// TIA Portal V16 program export: 0 tag tables, 0 data types, 2 data blocks, 11 code blocks (in call order from the OBs), 4 instance data blocks

DATA_BLOCK "DB_HMI"   // DB3
{ S7_Optimized_Access := 'TRUE' }
VERSION : 0.1
// stored: AutoNumber true, CodeModifiedDate 2020-02-26T07:38:35.2363514Z, CompileDate 2021-07-03T08:38:43.1466981Z, CreationDate 2020-02-26T07:38:17.5478271Z, DBAccessibleFromOPCUA true, DownloadWithoutReinit false, InterfaceModifiedDate 2020-02-26T07:38:35.2363514Z, IsConsistent true, IsKnowHowProtected false, IsOnlyStoredInLoadMemory false, IsPLCDB false, IsRetainMemResEnabled false, IsWriteProtectedInAS false, MemoryReserve 100, ModifiedDate 2020-02-26T07:38:35.2363514Z, ParameterModified 2020-02-26T07:38:35.2363514Z, StructureModified 2020-02-26T07:38:35.2363514Z
   VAR
      VlvLiq1 : "udtHMI_ValveControl";
      VlvLiq2 { S7_SetPoint := 'True'} : "udtHMI_ValveControl";
      VlvDrn { S7_SetPoint := 'True'} : "udtHMI_ValveControl";
   END_VAR
BEGIN
END_DATA_BLOCK

DATA_BLOCK "DB_ProgramLogic"   // DB4
{ S7_Optimized_Access := 'TRUE' }
VERSION : 0.1
// stored: AutoNumber true, CodeModifiedDate 2020-02-26T07:40:10.2847553Z, CompileDate 2021-07-03T08:38:37.7718266Z, CreationDate 2020-02-26T07:39:28.2364137Z, DBAccessibleFromOPCUA true, DownloadWithoutReinit false, InterfaceModifiedDate 2020-02-26T07:40:10.2847553Z, IsConsistent true, IsKnowHowProtected false, IsOnlyStoredInLoadMemory false, IsPLCDB false, IsRetainMemResEnabled false, IsWriteProtectedInAS false, MemoryReserve 100, ModifiedDate 2020-02-26T07:40:10.2847553Z, ParameterModified 2020-02-26T07:40:10.2847553Z, StructureModified 2020-02-26T07:40:10.2847553Z
   VAR
      VlvLiq1_Open : Bool;
      VlvLiq2_Open : Bool;
      VlvDrn_Open : Bool;
   END_VAR
BEGIN
END_DATA_BLOCK

ORGANIZATION_BLOCK "Main"   // OB1, FBD, ProgramCycle
TITLE = "Main Program Sweep (Cycle)"
{ S7_Optimized_Access := 'TRUE' }
VERSION : 0.1
// stored: AutoNumber true, CodeModifiedDate 2021-08-10T08:54:10.1985647Z, CompileDate 2021-08-10T08:57:18.4266346Z, ConstantName OB_Main, CreationDate 2020-02-26T07:01:34.5488912Z, EventClass Program cycle, HandleErrorsWithinBlock false, InterfaceModifiedDate 2008-07-21T16:55:08.419547Z, IsConsistent true, IsIECCheckEnabled false, IsKnowHowProtected false, IsWriteProtected false, ModifiedDate 2021-08-10T08:54:10.1985647Z, ParameterModified 2008-07-21T16:55:08.419547Z, PLCSimAdvancedSupport true, PriorityNumber 1, ProcessImagePartNumber 65535, SetENOAutomatically false, StructureModified 2008-07-21T16:55:08.419547Z
   VAR_INPUT
      Initial_Call : Bool;   // Initial call of this OB
      Remanence : Bool;   // =True, if remanent data are available
   END_VAR
BEGIN

REGION Network 1
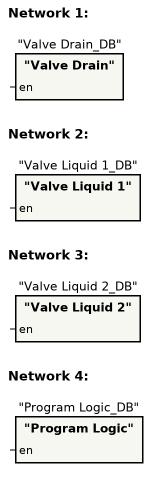
   "Valve Drain_DB"();   // "Valve Drain"
END_REGION

REGION Network 2
   "Valve Liquid 1_DB"();   // "Valve Liquid 1"
END_REGION

REGION Network 3
   "Valve Liquid 2_DB"();   // "Valve Liquid 2"
END_REGION

REGION Network 4
   "Program Logic_DB"();   // "Program Logic"
END_REGION
END_ORGANIZATION_BLOCK

FUNCTION_BLOCK "Valve Drain"   // FB4, FBD
{ S7_Optimized_Access := 'TRUE' }
VERSION : 0.1
// stored: AutoNumber true, CodeModifiedDate 2020-02-26T13:08:47.8951368Z, CompileDate 2021-07-03T08:38:43.4907825Z, CreationDate 2020-02-26T07:16:51.9541274Z, DownloadWithoutReinit false, HandleErrorsWithinBlock false, InterfaceModifiedDate 2020-02-26T12:48:59.514304Z, IsConsistent true, IsIECCheckEnabled false, IsKnowHowProtected false, ISMultiInstanceCapable true, IsRetainMemResEnabled false, IsWriteProtected false, LibraryConformanceStatus Warning: The object contains access to global data blocks. Warning: The block contains direct access to inputs, outputs, bit memories, indirect access to the registry or indirect access to external memory areas that are unknown at the time of compilation., MemoryReserve 100, ModifiedDate 2020-05-11T19:30:06.5567173Z, ParameterModified 2020-02-26T07:16:51.9541274Z, PLCSimAdvancedSupport true, SetENOAutomatically false, StructureModified 2020-02-26T12:48:59.514304Z, UDAEnableTagReadback false
   VAR
      VlvDrn : "fbValve_Solenoid";
   END_VAR
BEGIN

REGION Network 1
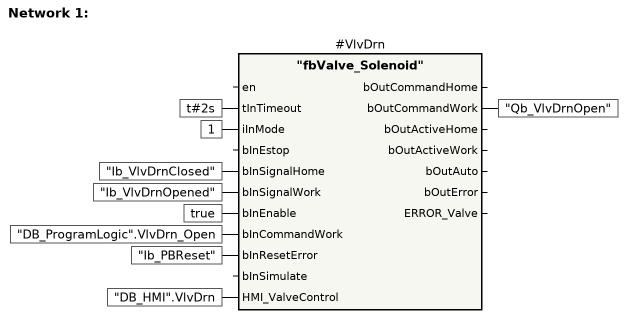
   #VlvDrn(tInTimeout := t#2s,   // "fbValve_Solenoid"
           iInMode := 1,
           bInSignalHome := "Ib_VlvDrnClosed",
           bInSignalWork := "Ib_VlvDrnOpened",
           bInEnable := true,
           bInCommandWork := "DB_ProgramLogic".VlvDrn_Open,
           bInResetError := "Ib_PBReset",
           HMI_ValveControl := "DB_HMI".VlvDrn,
           bOutCommandWork => "Qb_VlvDrnOpen");
END_REGION
END_FUNCTION_BLOCK

FUNCTION_BLOCK "fbValve_Solenoid"   // FB110, FBD
TITLE = Controls a double- or single-acting valve
{ S7_Optimized_Access := 'TRUE' }
VERSION : 0.1
// stored: AutoNumber false, CodeModifiedDate 2021-08-10T11:52:58.0273326Z, CompileDate 2021-08-10T11:53:23.0999729Z, CreationDate 2020-02-26T07:34:28.9567791Z, DownloadWithoutReinit false, HandleErrorsWithinBlock false, InterfaceModifiedDate 2019-07-17T06:42:37.7805928Z, IsConsistent true, IsIECCheckEnabled false, IsKnowHowProtected false, ISMultiInstanceCapable true, IsRetainMemResEnabled false, IsWriteProtected false, LibraryConformanceStatus Warning: The object contains access to global PLC constants., LibraryType fbValve_Solenoid V 3.0.6 in test, LibraryTypeVersionGuid 0a9fd967-cd2b-46e1-afc3-82055bb762c7, MemoryReserve 100, ModifiedDate 2021-08-10T11:52:58.0273326Z, ParameterModified 2019-07-17T06:42:37.7805928Z, PLCSimAdvancedSupport true, SetENOAutomatically false, StructureModified 2019-07-17T06:42:37.7805928Z, UDAEnableTagReadback false
   VAR_INPUT
      tInTimeout { ExternalAccessible := 'False'; ExternalVisible := 'False'; ExternalWritable := 'False'} : Time;   // Timeout time for an actuator's feedback to activate before giving a fault
      iInMode { ExternalAccessible := 'False'; ExternalVisible := 'False'; ExternalWritable := 'False'} : Int;   // Mode Selection
      bInEstop { ExternalAccessible := 'False'; ExternalVisible := 'False'; ExternalWritable := 'False'} : Bool;   // Estop
      bInSignalHome { ExternalAccessible := 'False'; ExternalVisible := 'False'; ExternalWritable := 'False'} : Bool;   // Home position feedback
      bInSignalWork { ExternalAccessible := 'False'; ExternalVisible := 'False'; ExternalWritable := 'False'} : Bool;   // Work position feedback
      bInEnable { ExternalAccessible := 'False'; ExternalVisible := 'False'; ExternalWritable := 'False'} : Bool;   // Home and Work Enabled
      bInCommandWork { ExternalAccessible := 'False'; ExternalVisible := 'False'; ExternalWritable := 'False'} : Bool;   // Move to work position in automatic mode
      bInResetError { ExternalAccessible := 'False'; ExternalVisible := 'False'; ExternalWritable := 'False'} : Bool;   // Reset Error
      bInSimulate { ExternalAccessible := 'False'; ExternalVisible := 'False'; ExternalWritable := 'False'} : Bool;   // Activate device simulation
   END_VAR
   VAR_OUTPUT
      bOutCommandHome { ExternalAccessible := 'False'; ExternalVisible := 'False'; ExternalWritable := 'False'} : Bool;   // Home position command
      bOutCommandWork { ExternalAccessible := 'False'; ExternalVisible := 'False'; ExternalWritable := 'False'} : Bool;   // Work position command
      bOutActiveHome { ExternalAccessible := 'False'; ExternalVisible := 'False'; ExternalWritable := 'False'} : Bool;   // Valve is in home position
      bOutActiveWork { ExternalAccessible := 'False'; ExternalVisible := 'False'; ExternalWritable := 'False'} : Bool;   // Valve is in work position
      bOutAuto { ExternalAccessible := 'False'; ExternalVisible := 'False'; ExternalWritable := 'False'} : Bool;   // Block in auto mode
      bOutError { ExternalAccessible := 'False'; ExternalVisible := 'False'; ExternalWritable := 'False'} : Bool;   // Error exists
      ERROR_Valve { ExternalAccessible := 'False'; ExternalVisible := 'False'; ExternalWritable := 'False'} : "udtError_Valve";   // Valve error structure
   END_VAR
   VAR_IN_OUT
      HMI_ValveControl : "udtHMI_ValveControl";   // HMI valve control
   END_VAR
   VAR
      ErrorScroller { ExternalAccessible := 'False'; ExternalVisible := 'False'; ExternalWritable := 'False'; S7_SetPoint := 'True'} : "fbErrorScroller";   // Sub-block to handle error scroller
      TON_TimeOut { ExternalAccessible := 'False'; ExternalVisible := 'False'; ExternalWritable := 'False'; S7_SetPoint := 'True'} : TON_TIME;   // Timer for Error Timeout
      iLastMode { ExternalAccessible := 'False'; ExternalVisible := 'False'; ExternalWritable := 'False'} : Int;   // Last mode code
      bNewMode { ExternalAccessible := 'False'; ExternalVisible := 'False'; ExternalWritable := 'False'} : Bool;   // New mode selected
      bEnableHome { ExternalAccessible := 'False'; ExternalVisible := 'False'; ExternalWritable := 'False'} : Bool;   // Home position enabled
      bEnableWork { ExternalAccessible := 'False'; ExternalVisible := 'False'; ExternalWritable := 'False'} : Bool;   // Work position enabled
      bAutoMode { ExternalAccessible := 'False'; ExternalVisible := 'False'; ExternalWritable := 'False'} : Bool;   // Auto Mode is active
      bManualMode { ExternalAccessible := 'False'; ExternalVisible := 'False'; ExternalWritable := 'False'} : Bool;   // Manual Mode is active
      bReset { ExternalAccessible := 'False'; ExternalVisible := 'False'; ExternalWritable := 'False'} : Bool;
      bTON_TimeOut { ExternalAccessible := 'False'; ExternalVisible := 'False'; ExternalWritable := 'False'} : Bool;
      bPB_Home { ExternalAccessible := 'False'; ExternalVisible := 'False'; ExternalWritable := 'False'} : Bool;
      bPB_Work { ExternalAccessible := 'False'; ExternalVisible := 'False'; ExternalWritable := 'False'} : Bool;
      bPB_ResetError { ExternalAccessible := 'False'; ExternalVisible := 'False'; ExternalWritable := 'False'} : Bool;
   END_VAR
   VAR_TEMP
      tTimeoutElapsed : Time;   // Elapsed time for TON_Timeout
      bTemp : Bool;
   END_VAR
   VAR_TEMP   // added for the SCL form of the ladder/FBD networks
      _w1 : Bool;
      _w2 : Bool;
   END_VAR
BEGIN

REGION Network 1: --------------------------------------------------------- Inputs ------------------------------------------------------------------
END_REGION

REGION Network 2: Read HMI input buttons
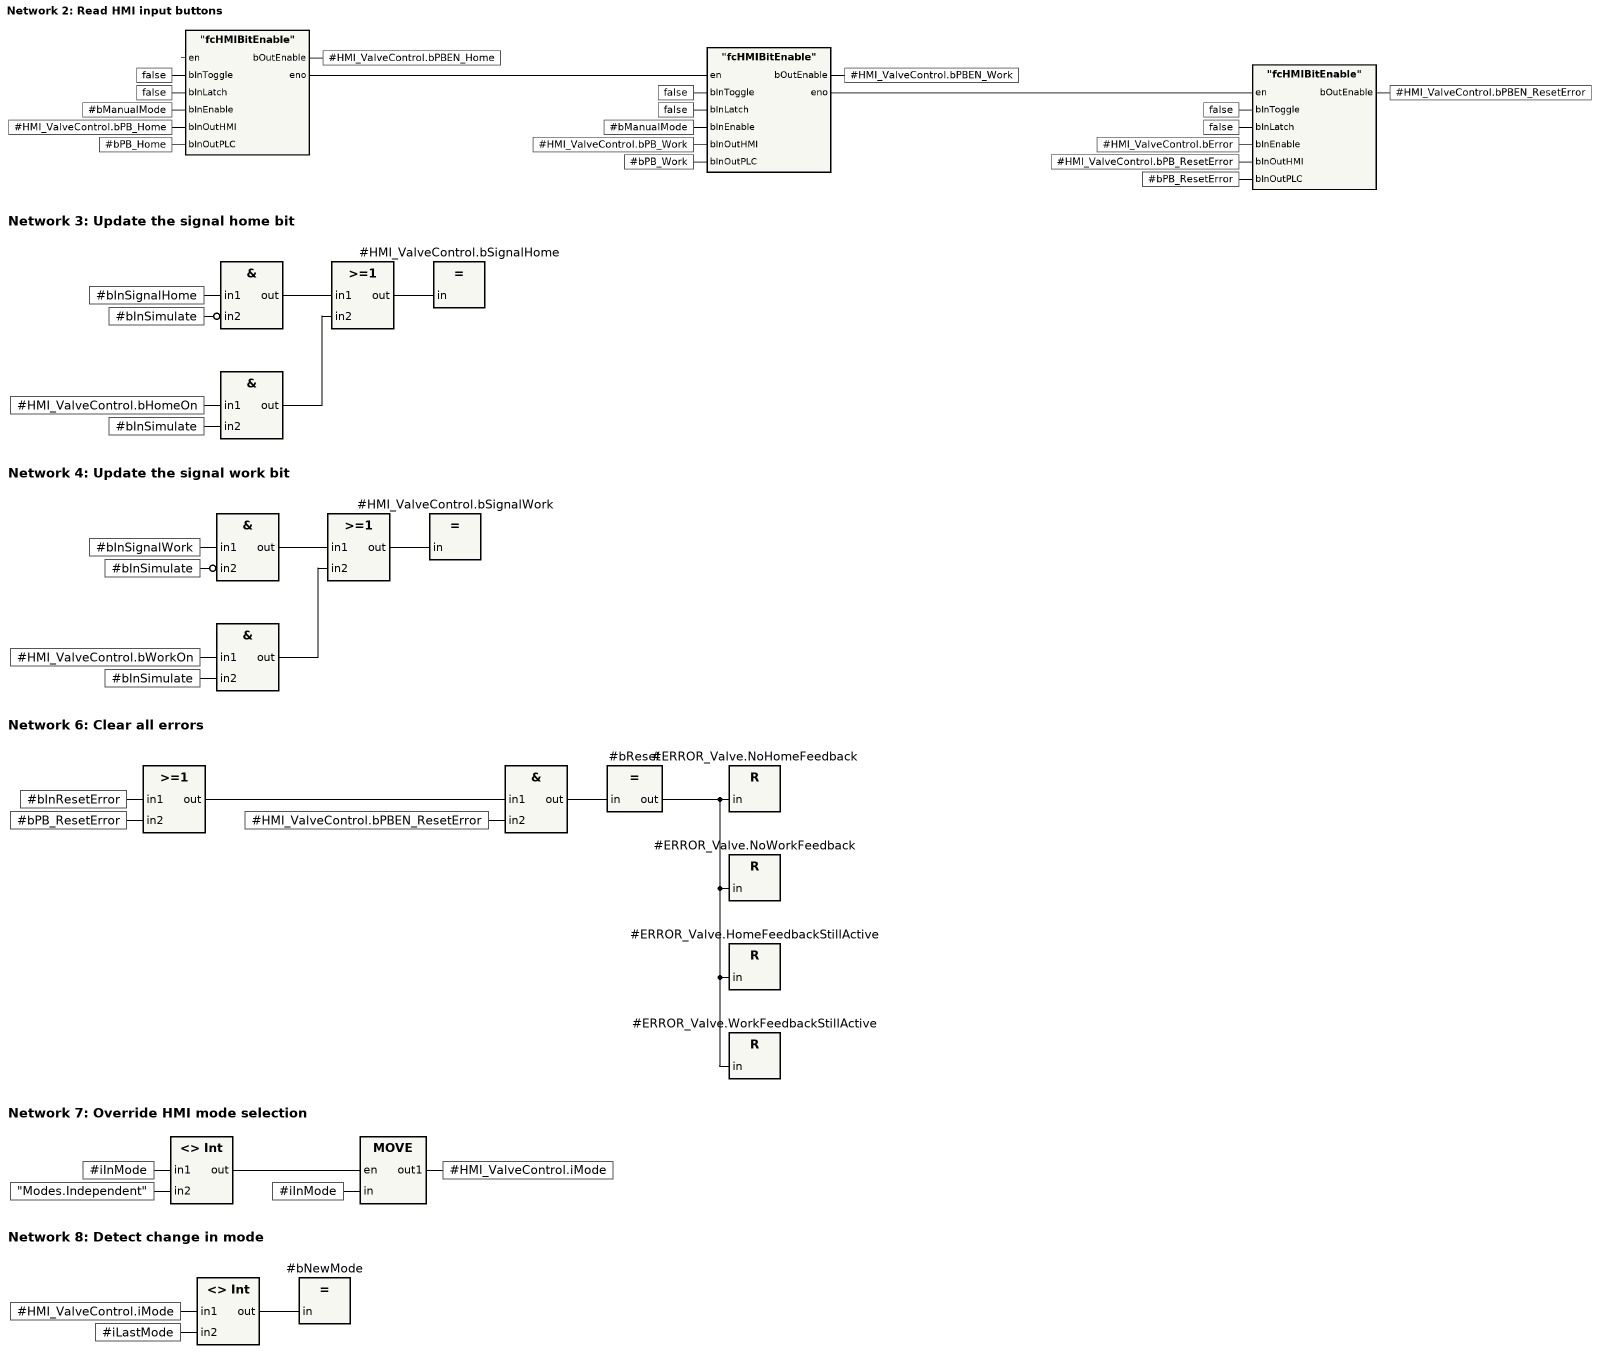
   "fcHMIBitEnable"(bInToggle := false,
                    bInLatch := false,
                    bInEnable := #bManualMode,
                    bInOutHMI := #HMI_ValveControl.bPB_Home,
                    bInOutPLC := #bPB_Home,
                    bOutEnable => #HMI_ValveControl.bPBEN_Home,
                    ENO => #_w1);
   "fcHMIBitEnable"(EN := #_w1,
                    bInToggle := false,
                    bInLatch := false,
                    bInEnable := #bManualMode,
                    bInOutHMI := #HMI_ValveControl.bPB_Work,
                    bInOutPLC := #bPB_Work,
                    bOutEnable => #HMI_ValveControl.bPBEN_Work,
                    ENO => #_w2);
   IF #_w2 THEN
       "fcHMIBitEnable"(bInToggle := false,
                        bInLatch := false,
                        bInEnable := #HMI_ValveControl.bError,
                        bInOutHMI := #HMI_ValveControl.bPB_ResetError,
                        bInOutPLC := #bPB_ResetError,
                        bOutEnable => #HMI_ValveControl.bPBEN_ResetError);
   END_IF;
END_REGION

REGION Network 3: Update the signal home bit
   #HMI_ValveControl.bSignalHome := (#bInSignalHome AND NOT #bInSimulate) OR (#HMI_ValveControl.bHomeOn AND #bInSimulate);
END_REGION

REGION Network 4: Update the signal work bit
   #HMI_ValveControl.bSignalWork := (#bInSignalWork AND NOT #bInSimulate) OR (#HMI_ValveControl.bWorkOn AND #bInSimulate);
END_REGION

REGION Network 5: --------------------------------------------------- Control Logic ------------------------------------------------------------
END_REGION

REGION Network 6: Clear all errors
   #bReset := (#bInResetError OR #bPB_ResetError) AND #HMI_ValveControl.bPBEN_ResetError;
   IF #bReset THEN
       #ERROR_Valve.NoHomeFeedback := FALSE;
       #ERROR_Valve.NoWorkFeedback := FALSE;
       #ERROR_Valve.HomeFeedbackStillActive := FALSE;
       #ERROR_Valve.WorkFeedbackStillActive := FALSE;
   END_IF;
END_REGION

REGION Network 7: Override HMI mode selection
   IF #iInMode <> "Modes.Independent" THEN #HMI_ValveControl.iMode := #iInMode; END_IF;
END_REGION

REGION Network 8: Detect change in mode
   #bNewMode := #HMI_ValveControl.iMode <> #iLastMode;
END_REGION

REGION Network 9: Keep track of last mode
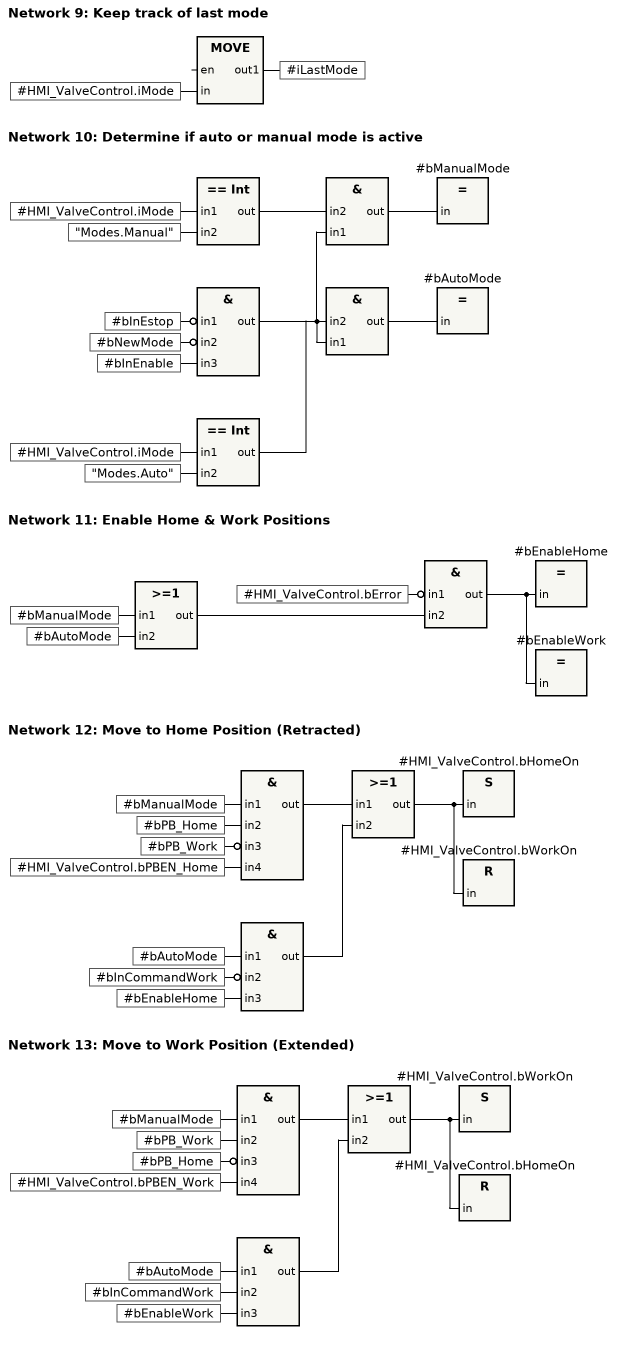
   #iLastMode := #HMI_ValveControl.iMode;
END_REGION

REGION Network 10: Determine if auto or manual mode is active
   #_w1 := NOT #bInEstop AND NOT #bNewMode AND #bInEnable;
   #bManualMode := (#HMI_ValveControl.iMode = "Modes.Manual") AND #_w1;
   #bAutoMode := (#HMI_ValveControl.iMode = "Modes.Auto") AND #_w1;
END_REGION

REGION Network 11: Enable Home & Work Positions
   // IF manual mode AND no estop AND not a new mode AND enabled => 
   // --if no cylinder errors, enable move to Home and Work
   // --enable home and work HMI buttons only in manual mode
   #bEnableHome := NOT #HMI_ValveControl.bError AND (#bManualMode OR #bAutoMode);
   #bEnableWork := #bEnableHome;
END_REGION

REGION Network 12: Move to Home Position (Retracted)
   // IF manual mode and home button is pressed =>
   // --Set close cylinder
   IF (#bManualMode AND #bPB_Home AND NOT #bPB_Work AND #HMI_ValveControl.bPBEN_Home) OR (#bAutoMode AND NOT #bInCommandWork AND #bEnableHome) THEN
       #HMI_ValveControl.bHomeOn := TRUE;
       #HMI_ValveControl.bWorkOn := FALSE;
   END_IF;
END_REGION

REGION Network 13: Move to Work Position (Extended)
   // IF manual mode and work button button is pressed =>
   // --Set open cylinder
   IF (#bManualMode AND #bPB_Work AND NOT #bPB_Home AND #HMI_ValveControl.bPBEN_Work) OR (#bAutoMode AND #bInCommandWork AND #bEnableWork) THEN
       #HMI_ValveControl.bWorkOn := TRUE;
       #HMI_ValveControl.bHomeOn := FALSE;
   END_IF;
END_REGION

REGION Network 14: Reset home on if not enabled
   // IF in auto AND home is not enabled => RESET home command
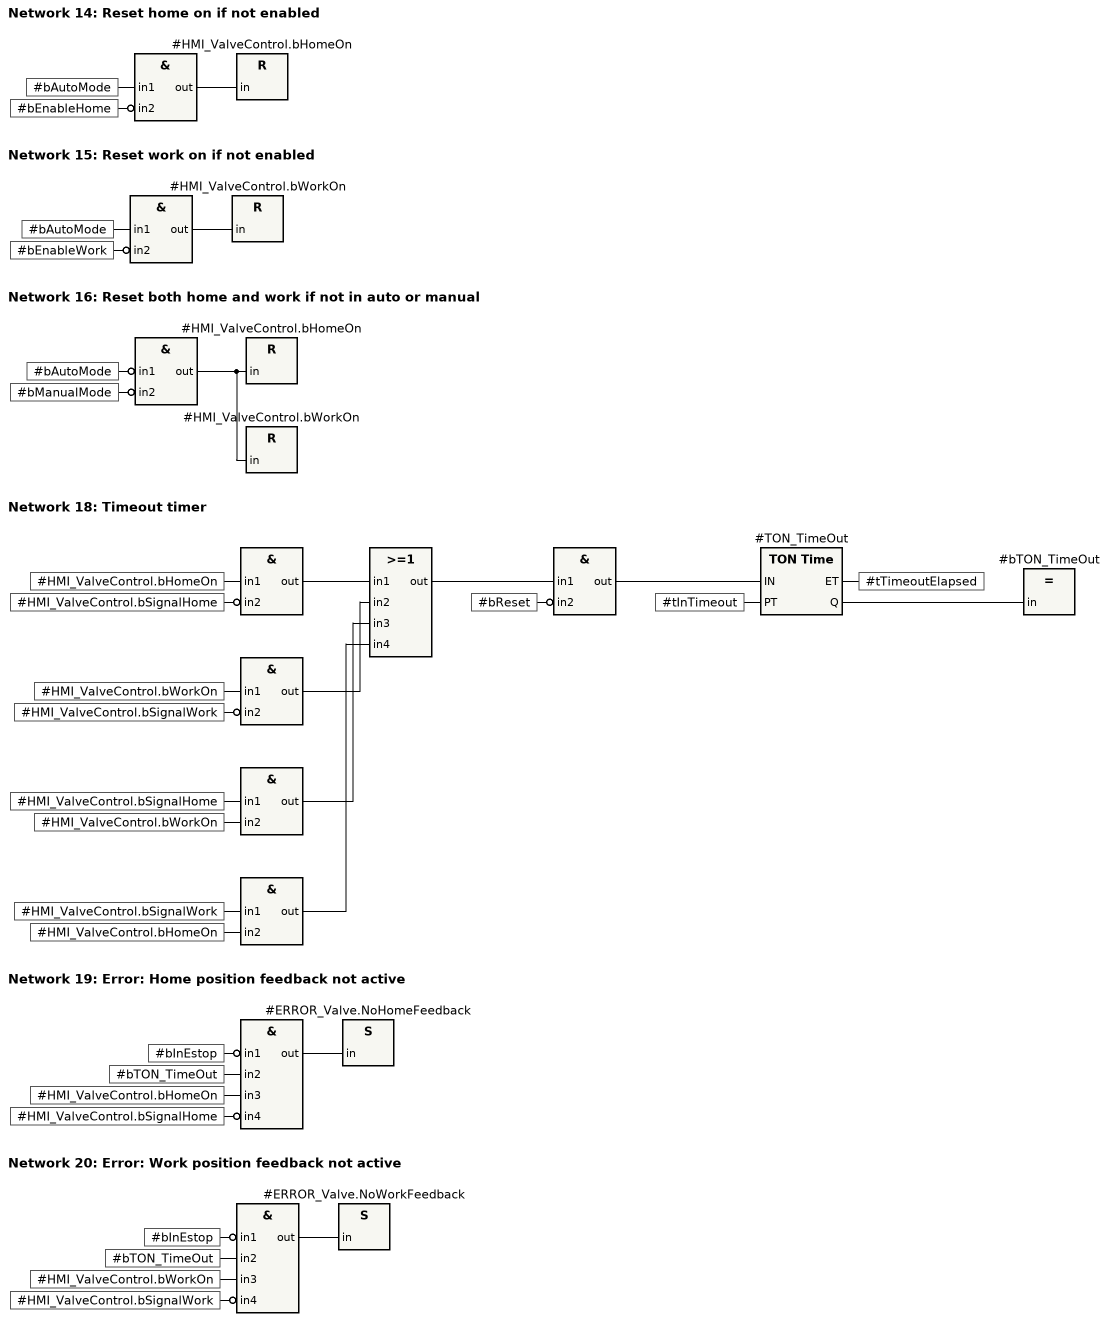
   IF #bAutoMode AND NOT #bEnableHome THEN #HMI_ValveControl.bHomeOn := FALSE; END_IF;
END_REGION

REGION Network 15: Reset work on if not enabled
   // IF in auto AND work is not enabled => RESET work command
   IF #bAutoMode AND NOT #bEnableWork THEN #HMI_ValveControl.bWorkOn := FALSE; END_IF;
END_REGION

REGION Network 16: Reset both home and work if not in auto or manual
   // IF not in auto AND not in manual => RESET home and work commands
   IF NOT #bAutoMode AND NOT #bManualMode THEN
       #HMI_ValveControl.bHomeOn := FALSE;
       #HMI_ValveControl.bWorkOn := FALSE;
   END_IF;
END_REGION

REGION Network 17: --------------------------------------------------------- Errors ------------------------------------------------------------------
END_REGION

REGION Network 18: Timeout timer
   // Time delay for errors
   #TON_TimeOut(IN := ((#HMI_ValveControl.bHomeOn AND NOT #HMI_ValveControl.bSignalHome) OR (#HMI_ValveControl.bWorkOn AND NOT #HMI_ValveControl.bSignalWork) OR (#HMI_ValveControl.bSignalHome AND #HMI_ValveControl.bWorkOn) OR (#HMI_ValveControl.bSignalWork AND #HMI_ValveControl.bHomeOn)) AND NOT #bReset,   // TON
                PT := #tInTimeout,
                ET => #tTimeoutElapsed);
   #bTON_TimeOut := #TON_TimeOut.Q;
END_REGION

REGION Network 19: Error: Home position feedback not active
   IF NOT #bInEstop AND #bTON_TimeOut AND #HMI_ValveControl.bHomeOn AND NOT #HMI_ValveControl.bSignalHome THEN
       #ERROR_Valve.NoHomeFeedback := TRUE;
   END_IF;
END_REGION

REGION Network 20: Error: Work position feedback not active
   // Not reach work position
   IF NOT #bInEstop AND #bTON_TimeOut AND #HMI_ValveControl.bWorkOn AND NOT #HMI_ValveControl.bSignalWork THEN
       #ERROR_Valve.NoWorkFeedback := TRUE;
   END_IF;
END_REGION

REGION Network 21: Error: Home position feedback still active
   // Home position still active
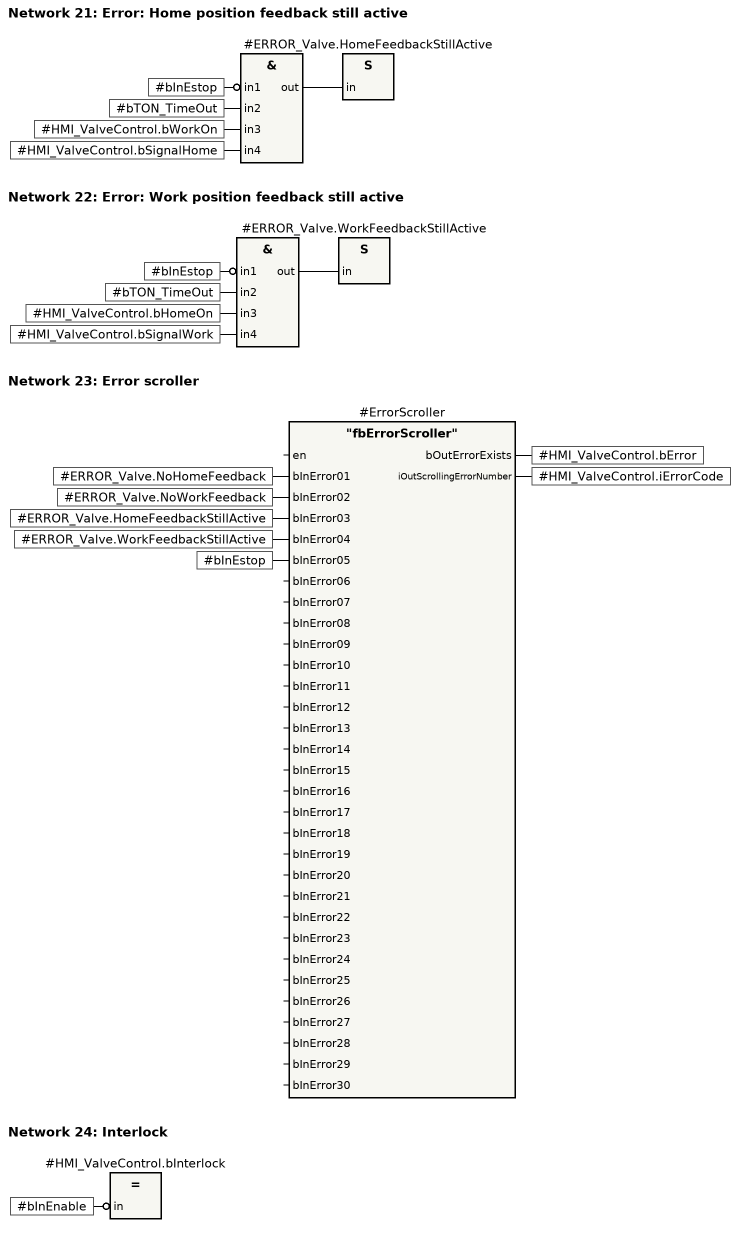
   IF NOT #bInEstop AND #bTON_TimeOut AND #HMI_ValveControl.bWorkOn AND #HMI_ValveControl.bSignalHome THEN
       #ERROR_Valve.HomeFeedbackStillActive := TRUE;
   END_IF;
END_REGION

REGION Network 22: Error: Work position feedback still active
   // Work position still active
   IF NOT #bInEstop AND #bTON_TimeOut AND #HMI_ValveControl.bHomeOn AND #HMI_ValveControl.bSignalWork THEN
       #ERROR_Valve.WorkFeedbackStillActive := TRUE;
   END_IF;
END_REGION

REGION Network 23: Error scroller
   // Call the Error-Scroller which cyles through all possible errors and checks 
   // their state for display on the HMI
   #ErrorScroller(bInError01 := #ERROR_Valve.NoHomeFeedback,   // "fbErrorScroller"
                  bInError02 := #ERROR_Valve.NoWorkFeedback,
                  bInError03 := #ERROR_Valve.HomeFeedbackStillActive,
                  bInError04 := #ERROR_Valve.WorkFeedbackStillActive,
                  bInError05 := #bInEstop,
                  bOutErrorExists => #HMI_ValveControl.bError,
                  iOutScrollingErrorNumber => #HMI_ValveControl.iErrorCode);
END_REGION

REGION Network 24: Interlock
   #HMI_ValveControl.bInterlock := NOT #bInEnable;
END_REGION

REGION Network 25: Set HMI status
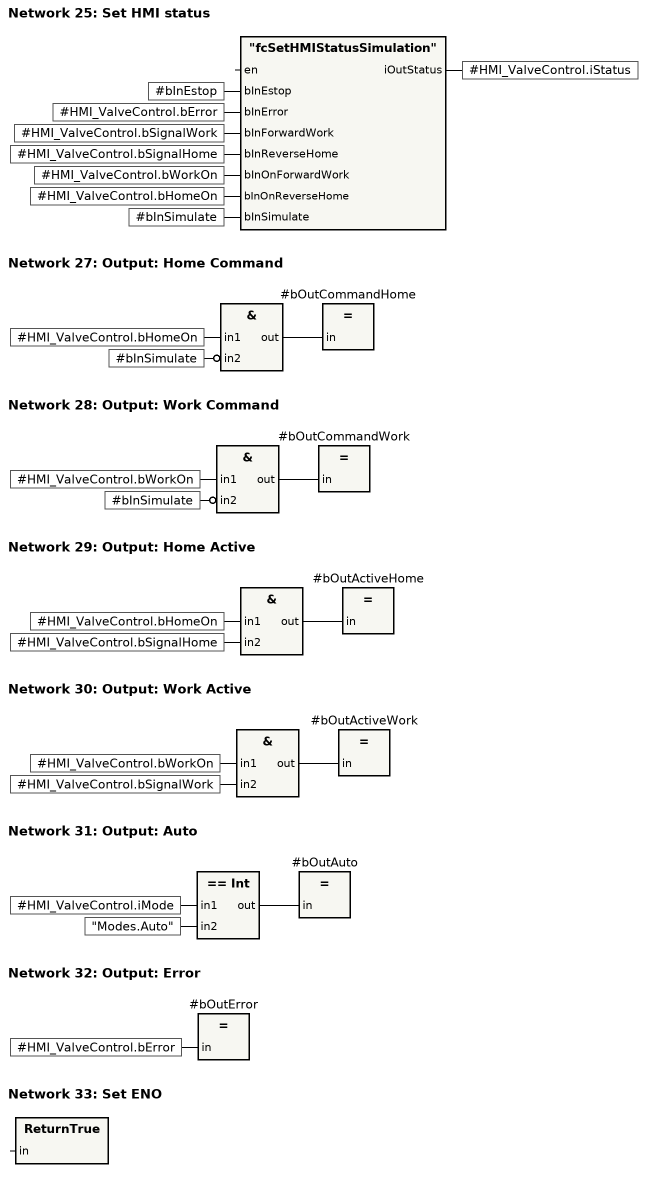
   "fcSetHMIStatusSimulation"(bInEstop := #bInEstop,
                           bInError := #HMI_ValveControl.bError,
                           bInForwardWork := #HMI_ValveControl.bSignalWork,
                           bInReverseHome := #HMI_ValveControl.bSignalHome,
                           bInOnForwardWork := #HMI_ValveControl.bWorkOn,
                           bInOnReverseHome := #HMI_ValveControl.bHomeOn,
                           bInSimulate := #bInSimulate,
                           iOutStatus => #HMI_ValveControl.iStatus);
END_REGION

REGION Network 26: -------------------------------------------------- Outputs --------------------------------------------------
END_REGION

REGION Network 27: Output: Home Command
   #bOutCommandHome := #HMI_ValveControl.bHomeOn AND NOT #bInSimulate;
END_REGION

REGION Network 28: Output: Work Command
   #bOutCommandWork := #HMI_ValveControl.bWorkOn AND NOT #bInSimulate;
END_REGION

REGION Network 29: Output: Home Active
   #bOutActiveHome := #HMI_ValveControl.bHomeOn AND #HMI_ValveControl.bSignalHome;
END_REGION

REGION Network 30: Output: Work Active
   #bOutActiveWork := #HMI_ValveControl.bWorkOn AND #HMI_ValveControl.bSignalWork;
END_REGION

REGION Network 31: Output: Auto
   #bOutAuto := #HMI_ValveControl.iMode = "Modes.Auto";
END_REGION

REGION Network 32: Output: Error
   #bOutError := #HMI_ValveControl.bError;
END_REGION

REGION Network 33: Set ENO
   ENO := TRUE;
   RETURN;
END_REGION
END_FUNCTION_BLOCK

FUNCTION "fcHMIBitEnable" : Void   // FC329, FBD
TITLE = Handles an async reading of an HMI bit to avoid race conditions, includes an enable bit
{ S7_Optimized_Access := 'TRUE' }
VERSION : 0.1
// stored: AutoNumber true, CodeModifiedDate 2020-08-01T14:00:25.8449031Z, CompileDate 2021-07-03T08:38:37.4904384Z, CreationDate 2020-02-26T07:34:28.9567791Z, HandleErrorsWithinBlock false, InterfaceModifiedDate 2017-10-26T17:33:11.2112674Z, IsConsistent true, IsIECCheckEnabled false, IsKnowHowProtected false, IsWriteProtected false, LibraryConformanceStatus The object is library-conformant., LibraryType fcHMIBitEnable V 3.0.3, LibraryTypeVersionGuid be26d641-fc92-415f-8b4f-76383b13c227, ModifiedDate 2020-08-01T14:00:32.9533133Z, ParameterModified 2017-10-26T17:33:11.2112674Z, PLCSimAdvancedSupport true, SetENOAutomatically false, StructureModified 2017-10-26T17:33:11.2112674Z, UDAEnableTagReadback false
   VAR_INPUT
      bInToggle : Bool;
      bInLatch : Bool;
      bInEnable : Bool;
   END_VAR
   VAR_OUTPUT
      bOutEnable : Bool;
   END_VAR
   VAR_IN_OUT
      bInOutHMI : Bool;
      bInOutPLC : Bool;
   END_VAR
   VAR_TEMP   // added for the SCL form of the ladder/FBD networks
      _w1 : Bool;
   END_VAR
BEGIN

REGION Network 1: If not latching or toggling, reset the PLC bit every scan
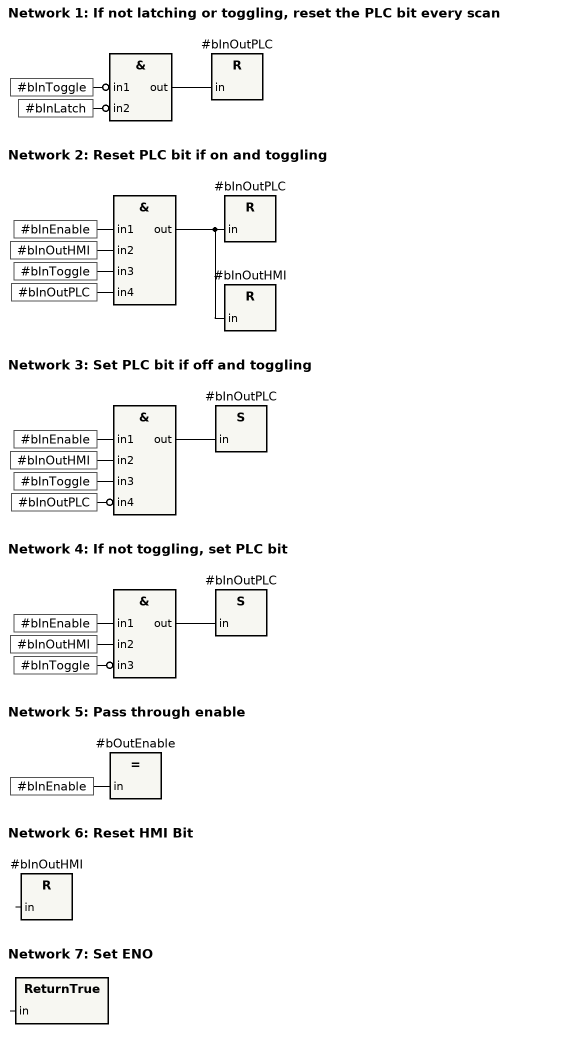
   IF NOT #bInToggle AND NOT #bInLatch THEN #bInOutPLC := FALSE; END_IF;
END_REGION

REGION Network 2: Reset PLC bit if on and toggling
   #_w1 := #bInEnable AND #bInOutHMI AND #bInToggle AND #bInOutPLC;
   IF #_w1 THEN
       #bInOutPLC := FALSE;
       #bInOutHMI := FALSE;
   END_IF;
END_REGION

REGION Network 3: Set PLC bit if off and toggling
   IF #bInEnable AND #bInOutHMI AND #bInToggle AND NOT #bInOutPLC THEN #bInOutPLC := TRUE; END_IF;
END_REGION

REGION Network 4: If not toggling, set PLC bit
   IF #bInEnable AND #bInOutHMI AND NOT #bInToggle THEN #bInOutPLC := TRUE; END_IF;
END_REGION

REGION Network 5: Pass through enable
   #bOutEnable := #bInEnable;
END_REGION

REGION Network 6: Reset HMI Bit
   #bInOutHMI := FALSE;
END_REGION

REGION Network 7: Set ENO
   ENO := TRUE;
   RETURN;
END_REGION
END_FUNCTION

FUNCTION_BLOCK "fbErrorScroller"   // FB330, FBD
TITLE = Scrolls through the error codes for display on the HMI
{ S7_Optimized_Access := 'TRUE' }
AUTHOR : DMC
FAMILY : Error
VERSION : 0.1
// stored: AutoNumber false, CodeModifiedDate 2020-08-01T14:01:08.1418864Z, CompileDate 2021-07-03T08:38:41.9599271Z, CreationDate 2020-02-26T07:34:28.9567791Z, DownloadWithoutReinit false, HandleErrorsWithinBlock false, InterfaceModifiedDate 2017-09-27T20:48:31.926835Z, IsConsistent true, IsIECCheckEnabled false, IsKnowHowProtected false, ISMultiInstanceCapable true, IsRetainMemResEnabled false, IsWriteProtected false, LibraryConformanceStatus The object is library-conformant., LibraryType fbErrorScroller V 3.0.3, LibraryTypeVersionGuid 88980ab5-f3a6-4351-a374-4d1b01e00ab7, MemoryReserve 100, ModifiedDate 2020-08-01T14:01:12.2238964Z, ParameterModified 2016-08-18T17:27:42.6947226Z, PLCSimAdvancedSupport true, SetENOAutomatically false, StructureModified 2016-12-19T18:48:15.4564605Z, UDAEnableTagReadback false
   VAR_INPUT
      bInError01 { ExternalAccessible := 'False'; ExternalVisible := 'False'; ExternalWritable := 'False'} : Bool;   // Error 1 In Error Array
      bInError02 { ExternalAccessible := 'False'; ExternalVisible := 'False'; ExternalWritable := 'False'} : Bool;   // Error 2 In Error Array
      bInError03 { ExternalAccessible := 'False'; ExternalVisible := 'False'; ExternalWritable := 'False'} : Bool;   // Error 3 In Error Array
      bInError04 { ExternalAccessible := 'False'; ExternalVisible := 'False'; ExternalWritable := 'False'} : Bool;   // Error 4 In Error Array
      bInError05 { ExternalAccessible := 'False'; ExternalVisible := 'False'; ExternalWritable := 'False'} : Bool;   // Error 5 In Error Array
      bInError06 { ExternalAccessible := 'False'; ExternalVisible := 'False'; ExternalWritable := 'False'} : Bool;   // Error 6 In Error Array
      bInError07 { ExternalAccessible := 'False'; ExternalVisible := 'False'; ExternalWritable := 'False'} : Bool;   // Error 7 In Error Array
      bInError08 { ExternalAccessible := 'False'; ExternalVisible := 'False'; ExternalWritable := 'False'} : Bool;   // Error 8 In Error Array
      bInError09 { ExternalAccessible := 'False'; ExternalVisible := 'False'; ExternalWritable := 'False'} : Bool;   // Error 9 In Error Array
      bInError10 { ExternalAccessible := 'False'; ExternalVisible := 'False'; ExternalWritable := 'False'} : Bool;   // Error 10 In Error Array
      bInError11 { ExternalAccessible := 'False'; ExternalVisible := 'False'; ExternalWritable := 'False'} : Bool;   // Error 11 In Error Array
      bInError12 { ExternalAccessible := 'False'; ExternalVisible := 'False'; ExternalWritable := 'False'} : Bool;   // Error 12 In Error Array
      bInError13 { ExternalAccessible := 'False'; ExternalVisible := 'False'; ExternalWritable := 'False'} : Bool;   // Error 13 In Error Array
      bInError14 { ExternalAccessible := 'False'; ExternalVisible := 'False'; ExternalWritable := 'False'} : Bool;   // Error 14 In Error Array
      bInError15 { ExternalAccessible := 'False'; ExternalVisible := 'False'; ExternalWritable := 'False'} : Bool;   // Error 15 In Error Array
      bInError16 { ExternalAccessible := 'False'; ExternalVisible := 'False'; ExternalWritable := 'False'} : Bool;   // Error 16 In Error Array
      bInError17 { ExternalAccessible := 'False'; ExternalVisible := 'False'; ExternalWritable := 'False'} : Bool;   // Error 17 In Error Array
      bInError18 { ExternalAccessible := 'False'; ExternalVisible := 'False'; ExternalWritable := 'False'} : Bool;   // Error 18 In Error Array
      bInError19 { ExternalAccessible := 'False'; ExternalVisible := 'False'; ExternalWritable := 'False'} : Bool;   // Error 19 In Error Array
      bInError20 { ExternalAccessible := 'False'; ExternalVisible := 'False'; ExternalWritable := 'False'} : Bool;   // Error 20 In Error Array
      bInError21 { ExternalAccessible := 'False'; ExternalVisible := 'False'; ExternalWritable := 'False'} : Bool;   // Error 21 In Error Array
      bInError22 { ExternalAccessible := 'False'; ExternalVisible := 'False'; ExternalWritable := 'False'} : Bool;   // Error 22 In Error Array
      bInError23 { ExternalAccessible := 'False'; ExternalVisible := 'False'; ExternalWritable := 'False'} : Bool;   // Error 23 In Error Array
      bInError24 { ExternalAccessible := 'False'; ExternalVisible := 'False'; ExternalWritable := 'False'} : Bool;   // Error 24 In Error Array
      bInError25 { ExternalAccessible := 'False'; ExternalVisible := 'False'; ExternalWritable := 'False'} : Bool;   // Error 25 In Error Array
      bInError26 { ExternalAccessible := 'False'; ExternalVisible := 'False'; ExternalWritable := 'False'} : Bool;   // Error 26 In Error Array
      bInError27 { ExternalAccessible := 'False'; ExternalVisible := 'False'; ExternalWritable := 'False'} : Bool;   // Error 27 In Error Array
      bInError28 { ExternalAccessible := 'False'; ExternalVisible := 'False'; ExternalWritable := 'False'} : Bool;   // Error 28 In Error Array
      bInError29 { ExternalAccessible := 'False'; ExternalVisible := 'False'; ExternalWritable := 'False'} : Bool;   // Error 29 In Error Array
      bInError30 { ExternalAccessible := 'False'; ExternalVisible := 'False'; ExternalWritable := 'False'} : Bool;   // Error 30 In Error Array
   END_VAR
   VAR_OUTPUT
      bOutErrorExists { ExternalAccessible := 'False'; ExternalVisible := 'False'; ExternalWritable := 'False'} : Bool;   // An Error Exists
      iOutScrollingErrorNumber { ExternalAccessible := 'False'; ExternalVisible := 'False'; ExternalWritable := 'False'} : Int;   // Current Index when scrolling through errors
   END_VAR
   VAR
      TON_ErrorDelay { ExternalAccessible := 'False'; ExternalVisible := 'False'; ExternalWritable := 'False'; S7_SetPoint := 'True'} : TON_TIME;   // Delay between each scroll for a new error
   END_VAR
   VAR DB_SPECIFIC
      abErrors { ExternalAccessible := 'False'; ExternalVisible := 'False'; ExternalWritable := 'False'} : Array[#ciIndexLow..#ciIndexHigh] of Bool;
   END_VAR
   VAR
      iNextScrollNum { ExternalAccessible := 'False'; ExternalVisible := 'False'; ExternalWritable := 'False'} : Int := 1;   // Index of next error position
      iErrorsScrollNum { ExternalAccessible := 'False'; ExternalVisible := 'False'; ExternalWritable := 'False'} : Int := 1;   // Index of current error position
      bScrolling { ExternalAccessible := 'False'; ExternalVisible := 'False'; ExternalWritable := 'False'} : Bool;   // Indicates we are scrolling
      bTON_ErrorDelay { ExternalAccessible := 'False'; ExternalVisible := 'False'; ExternalWritable := 'False'} : Bool;
   END_VAR
   VAR_TEMP
      bErrorExists : Bool;   // Error Exists
   END_VAR
   VAR CONSTANT
      ciNoErrrors : Int := 0;
      ciIndexLow : Int := 1;
      ciIndexHigh : Int := 30;
   END_VAR
   VAR_TEMP   // added for the SCL form of the ladder/FBD networks
      _w1 : Bool;
   END_VAR
BEGIN

REGION Network 1: Check for valid array indexes
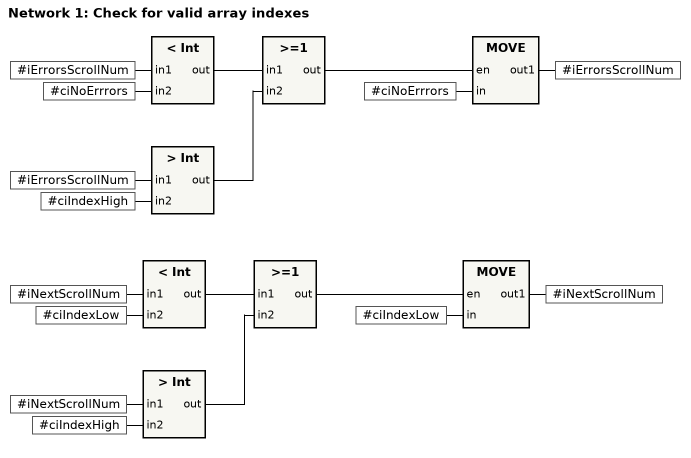
   IF (#iErrorsScrollNum < #ciNoErrrors) OR (#iErrorsScrollNum > #ciIndexHigh) THEN
       #iErrorsScrollNum := #ciNoErrrors;
   END_IF;
   IF (#iNextScrollNum < #ciIndexLow) OR (#iNextScrollNum > #ciIndexHigh) THEN
       #iNextScrollNum := #ciIndexLow;
   END_IF;
END_REGION

REGION Network 2: Check if error exists
   // OR all of the possible errors. If any error Exists, SET bErrorExists
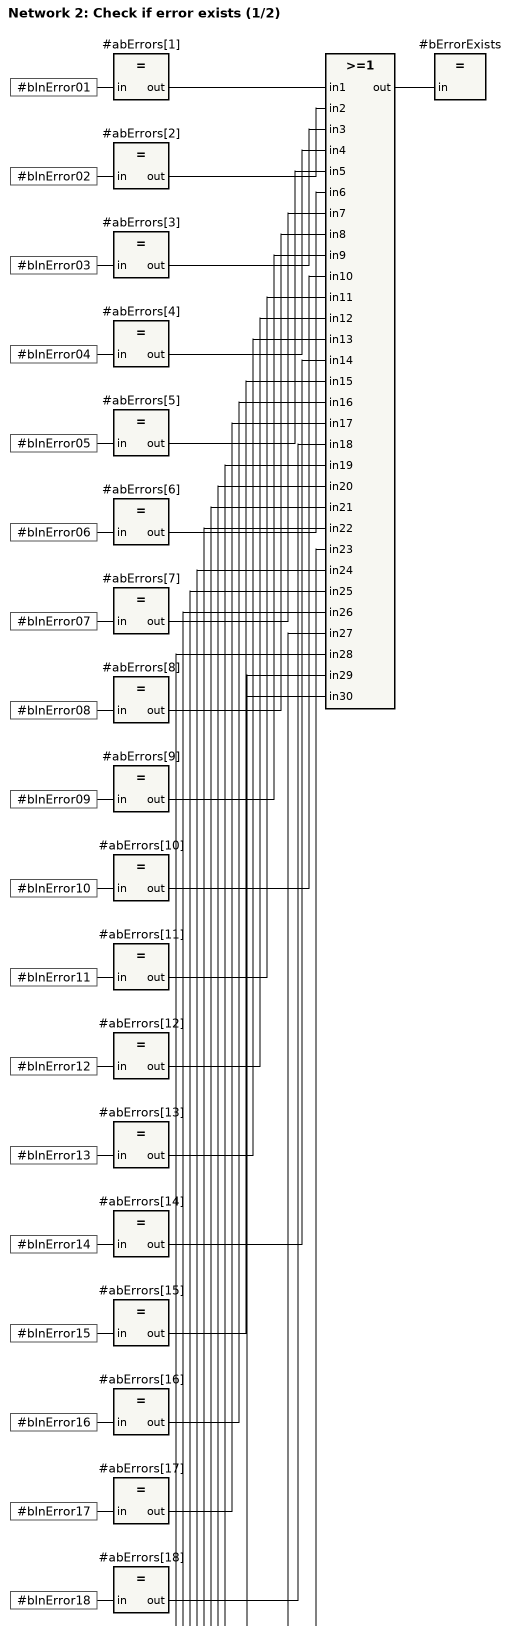
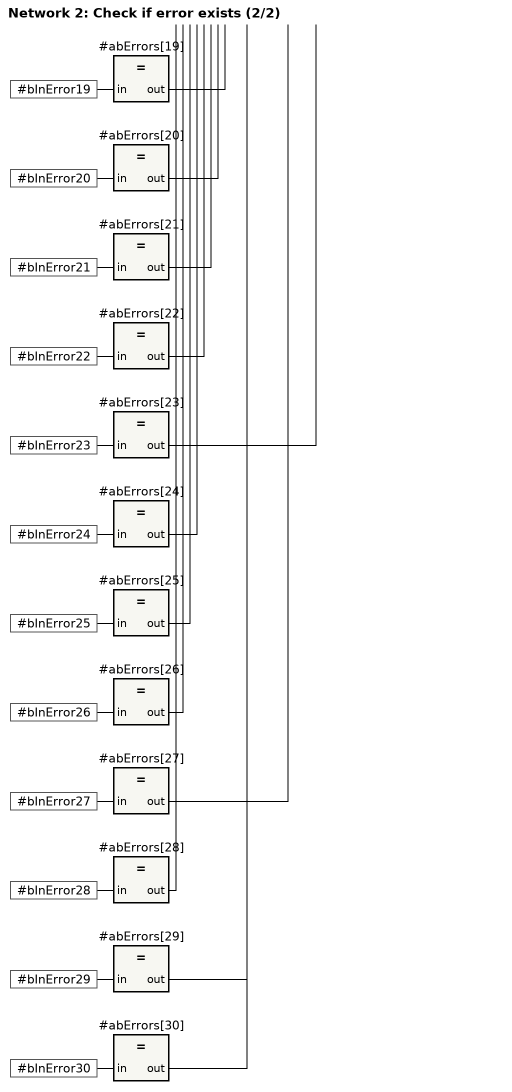
   #abErrors[1] := #bInError01;
   #abErrors[2] := #bInError02;
   #abErrors[3] := #bInError03;
   #abErrors[4] := #bInError04;
   #abErrors[5] := #bInError05;
   #abErrors[6] := #bInError06;
   #abErrors[7] := #bInError07;
   #abErrors[8] := #bInError08;
   #abErrors[9] := #bInError09;
   #abErrors[10] := #bInError10;
   #abErrors[11] := #bInError11;
   #abErrors[12] := #bInError12;
   #abErrors[13] := #bInError13;
   #abErrors[14] := #bInError14;
   #abErrors[15] := #bInError15;
   #abErrors[16] := #bInError16;
   #abErrors[17] := #bInError17;
   #abErrors[18] := #bInError18;
   #abErrors[19] := #bInError19;
   #abErrors[20] := #bInError20;
   #abErrors[21] := #bInError21;
   #abErrors[22] := #bInError22;
   #abErrors[23] := #bInError23;
   #abErrors[24] := #bInError24;
   #abErrors[25] := #bInError25;
   #abErrors[26] := #bInError26;
   #abErrors[27] := #bInError27;
   #abErrors[28] := #bInError28;
   #abErrors[29] := #bInError29;
   #abErrors[30] := #bInError30;
   #bErrorExists := #bInError01 OR #bInError02 OR #bInError03 OR #bInError04 OR #bInError05 OR #bInError06 OR #bInError07 OR #bInError08 OR #bInError09 OR #bInError10 OR #bInError11 OR #bInError12 OR #bInError13 OR #bInError14 OR #bInError15 OR #bInError16 OR #bInError17 OR #bInError18 OR #bInError19 OR #bInError20 OR #bInError21 OR #bInError22 OR #bInError23 OR #bInError24 OR #bInError25 OR #bInError26 OR #bInError27 OR #bInError28 OR #bInError29 OR #bInError30;
END_REGION

REGION Network 3: Timer to change displayed error
   // ============================ Scroll errors on HMI ========================
   // Timed delay
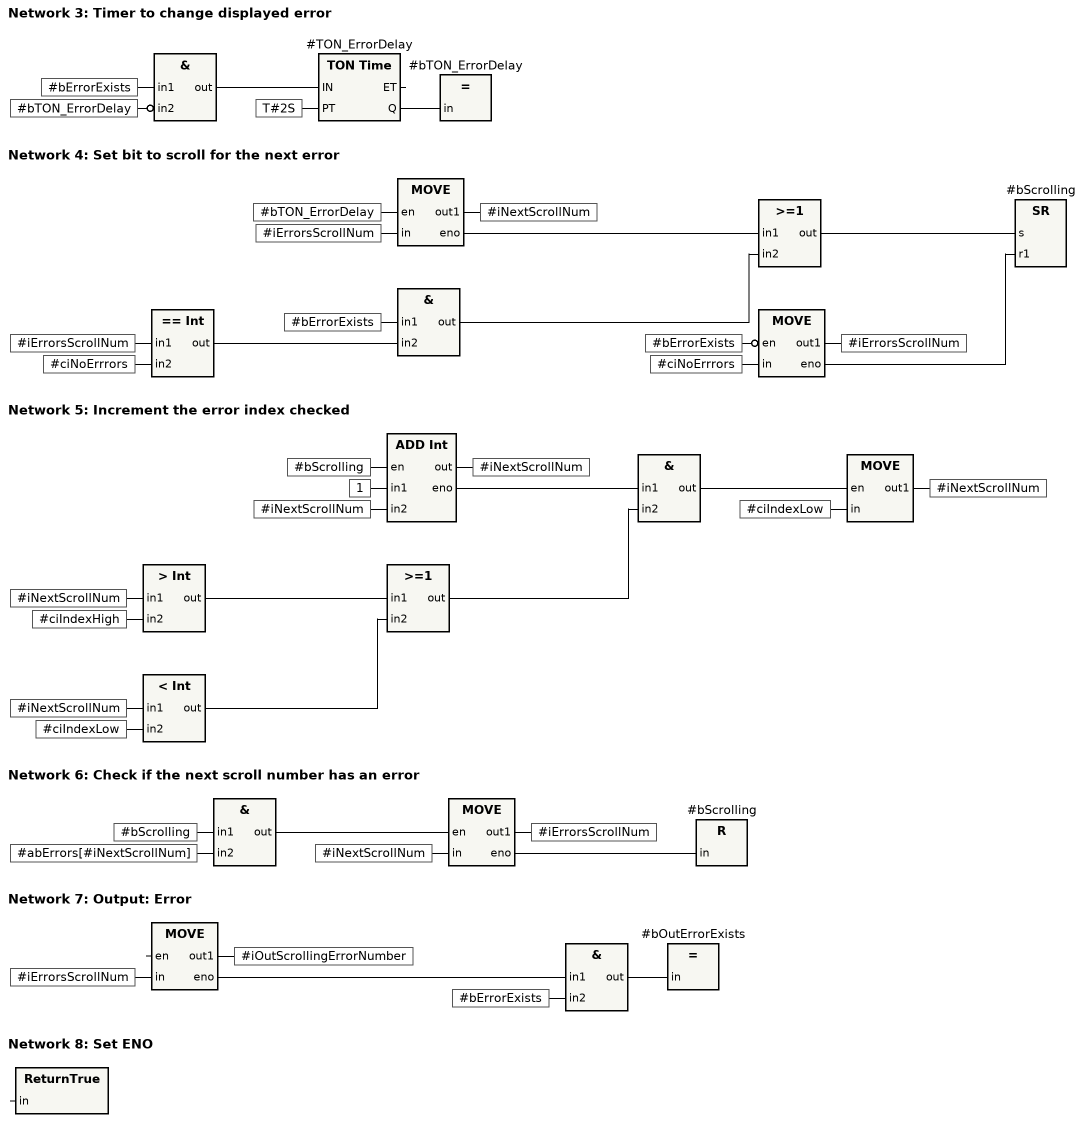
   #TON_ErrorDelay(IN := #bErrorExists AND NOT #bTON_ErrorDelay, PT := T#2S);   // TON
   #bTON_ErrorDelay := #TON_ErrorDelay.Q;
END_REGION

REGION Network 4: Set bit to scroll for the next error
   // Set a static bit indicating that we are scrolling.  
   // Each pass cycle through the function, we will increment.  
   // If there is no error, set the scroll num to 0 and turn off scrolling.  
   // It scrolls to an error immediately when an error occurs.
   // ENO of a box is taken as its EN; it also drops when the box reports an error
   IF #bTON_ErrorDelay THEN #iNextScrollNum := #iErrorsScrollNum; END_IF;
   #_w1 := #bTON_ErrorDelay OR (#bErrorExists AND (#iErrorsScrollNum = #ciNoErrrors));
   IF NOT #bErrorExists THEN #iErrorsScrollNum := #ciNoErrrors; END_IF;
   IF #_w1 THEN
       #bScrolling := TRUE;   // SR flip-flop
   END_IF;
   IF NOT #bErrorExists THEN #bScrolling := FALSE; END_IF;
END_REGION

REGION Network 5: Increment the error index checked
   // The function will only increment the scroll num one value per scan.  
   // It will scroll until it finds the next active error, then stop scrolling.  
   // Roll iNextScrollNum to 0 if it exceeds 30.
   // ENO of a box is taken as its EN; it also drops when the box reports an error
   IF #bScrolling THEN #iNextScrollNum := 1 + #iNextScrollNum; END_IF;
   IF #bScrolling AND ((#iNextScrollNum > #ciIndexHigh) OR (#iNextScrollNum < #ciIndexLow)) THEN
       #iNextScrollNum := #ciIndexLow;
   END_IF;
END_REGION

REGION Network 6: Check if the next scroll number has an error
   // If we found an error, stop scrolling.
   // ENO of a box is taken as its EN; it also drops when the box reports an error
   IF #bScrolling AND #abErrors[#iNextScrollNum] THEN
       #iErrorsScrollNum := #iNextScrollNum;
       #bScrolling := FALSE;
   END_IF;
END_REGION

REGION Network 7: Output: Error
   // Output the index of the error that exists.
   // ENO of a box is taken as its EN; it also drops when the box reports an error
   #iOutScrollingErrorNumber := #iErrorsScrollNum;
   #bOutErrorExists := #bErrorExists;
END_REGION

REGION Network 8: Set ENO
   ENO := TRUE;
   RETURN;
END_REGION
END_FUNCTION_BLOCK

FUNCTION "fcSetHMIStatusSimulation" : Void   // FC333, FBD
TITLE = Sets HMI Status
{ S7_Optimized_Access := 'TRUE' }
VERSION : 0.1
// Wrapper function for setting the HMI status of a device
// 
// In order of priority:
// 1. E-stop
// 2. Error
// 3. Forward/Work Position
// 4. Reverse/Home Position
// 5. Forward/Work On
// 6. Reverse/Home On
// 7. None
// stored: AutoNumber true, CodeModifiedDate 2020-08-01T14:00:45.2523905Z, CompileDate 2021-07-03T08:38:37.6631079Z, CreationDate 2020-02-26T07:34:28.9567791Z, HandleErrorsWithinBlock false, InterfaceModifiedDate 2019-07-16T09:38:07.8023625Z, IsConsistent true, IsIECCheckEnabled false, IsKnowHowProtected false, IsWriteProtected false, LibraryConformanceStatus Warning: The object contains access to global PLC constants., LibraryType fcSetHMIStatusSimulation V 3.0.4, LibraryTypeVersionGuid 66f3681c-ca78-4b7d-9ef9-bd50d3b993d6, ModifiedDate 2020-08-01T14:00:53.126388Z, ParameterModified 2019-07-16T09:38:07.8023625Z, PLCSimAdvancedSupport true, SetENOAutomatically false, StructureModified 2019-07-16T09:38:07.8023625Z, UDAEnableTagReadback false
   VAR_INPUT
      bInEstop : Bool;
      bInError : Bool;
      bInForwardWork : Bool;
      bInReverseHome : Bool;
      bInOnForwardWork : Bool;
      bInOnReverseHome : Bool;
      bInSimulate : Bool;
   END_VAR
   VAR_OUTPUT
      iOutStatus : Int;
   END_VAR
BEGIN

REGION Network 1: Set Reverse/Home On
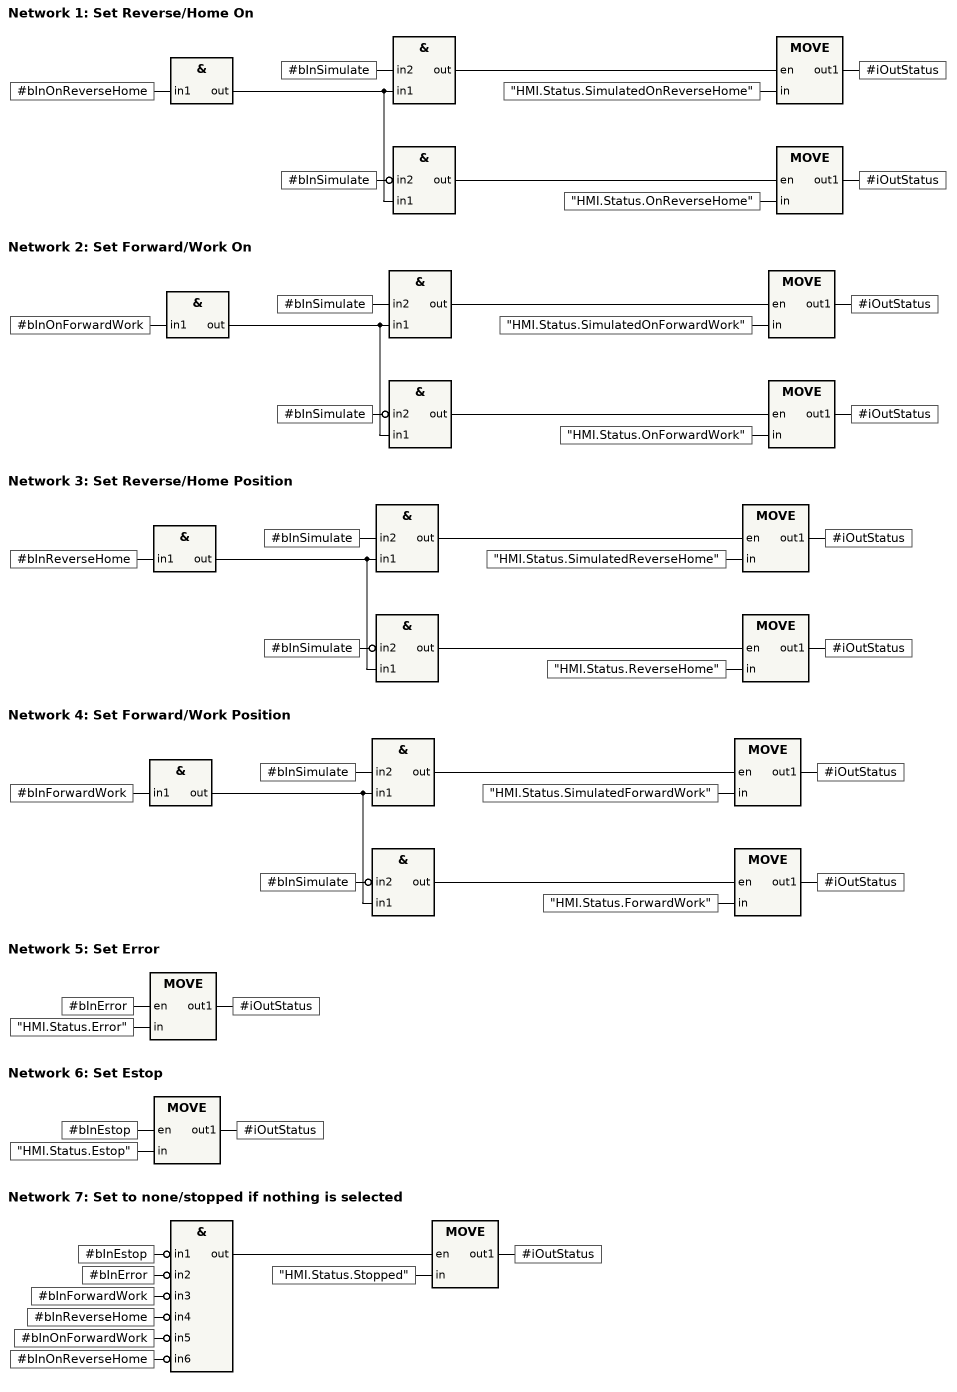
   IF #bInSimulate AND #bInOnReverseHome THEN #iOutStatus := "HMI.Status.SimulatedOnReverseHome"; END_IF;
   IF NOT #bInSimulate AND #bInOnReverseHome THEN #iOutStatus := "HMI.Status.OnReverseHome"; END_IF;
END_REGION

REGION Network 2: Set Forward/Work On
   IF #bInSimulate AND #bInOnForwardWork THEN #iOutStatus := "HMI.Status.SimulatedOnForwardWork"; END_IF;
   IF NOT #bInSimulate AND #bInOnForwardWork THEN #iOutStatus := "HMI.Status.OnForwardWork"; END_IF;
END_REGION

REGION Network 3: Set Reverse/Home Position
   IF #bInSimulate AND #bInReverseHome THEN #iOutStatus := "HMI.Status.SimulatedReverseHome"; END_IF;
   IF NOT #bInSimulate AND #bInReverseHome THEN #iOutStatus := "HMI.Status.ReverseHome"; END_IF;
END_REGION

REGION Network 4: Set Forward/Work Position
   IF #bInSimulate AND #bInForwardWork THEN #iOutStatus := "HMI.Status.SimulatedForwardWork"; END_IF;
   IF NOT #bInSimulate AND #bInForwardWork THEN #iOutStatus := "HMI.Status.ForwardWork"; END_IF;
END_REGION

REGION Network 5: Set Error
   IF #bInError THEN #iOutStatus := "HMI.Status.Error"; END_IF;
END_REGION

REGION Network 6: Set Estop
   IF #bInEstop THEN #iOutStatus := "HMI.Status.Estop"; END_IF;
END_REGION

REGION Network 7: Set to none/stopped if nothing is selected
   IF NOT #bInEstop AND NOT #bInError AND NOT #bInForwardWork AND NOT #bInReverseHome AND NOT #bInOnForwardWork AND NOT #bInOnReverseHome THEN
       #iOutStatus := "HMI.Status.Stopped";
   END_IF;
END_REGION

REGION Network 8: Set ENO
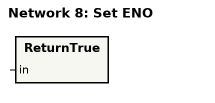
   ENO := TRUE;
   RETURN;
END_REGION
END_FUNCTION

FUNCTION_BLOCK "Valve Liquid 1"   // FB2, FBD
{ S7_Optimized_Access := 'TRUE' }
VERSION : 0.1
// stored: AutoNumber true, CodeModifiedDate 2020-02-26T13:08:56.9440303Z, CompileDate 2021-07-03T08:38:43.1627385Z, CreationDate 2020-02-26T07:16:31.1886327Z, DownloadWithoutReinit false, HandleErrorsWithinBlock false, InterfaceModifiedDate 2020-02-26T12:49:32.479094Z, IsConsistent true, IsIECCheckEnabled false, IsKnowHowProtected false, ISMultiInstanceCapable true, IsRetainMemResEnabled false, IsWriteProtected false, LibraryConformanceStatus Warning: The object contains access to global data blocks. Warning: The block contains direct access to inputs, outputs, bit memories, indirect access to the registry or indirect access to external memory areas that are unknown at the time of compilation., MemoryReserve 100, ModifiedDate 2020-02-26T13:08:56.9440303Z, ParameterModified 2020-02-26T07:16:31.1886327Z, PLCSimAdvancedSupport true, SetENOAutomatically false, StructureModified 2020-02-26T12:49:32.479094Z, UDAEnableTagReadback false
   VAR
      VlvLiq1 : "fbValve_Solenoid";
   END_VAR
BEGIN

REGION Network 1
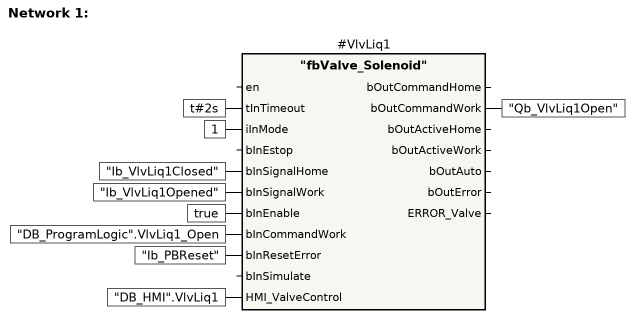
   #VlvLiq1(tInTimeout := t#2s,   // "fbValve_Solenoid"
            iInMode := 1,
            bInSignalHome := "Ib_VlvLiq1Closed",
            bInSignalWork := "Ib_VlvLiq1Opened",
            bInEnable := true,
            bInCommandWork := "DB_ProgramLogic".VlvLiq1_Open,
            bInResetError := "Ib_PBReset",
            HMI_ValveControl := "DB_HMI".VlvLiq1,
            bOutCommandWork => "Qb_VlvLiq1Open");
END_REGION
END_FUNCTION_BLOCK

FUNCTION_BLOCK "Valve Liquid 2"   // FB3, FBD
{ S7_Optimized_Access := 'TRUE' }
VERSION : 0.1
// stored: AutoNumber true, CodeModifiedDate 2020-02-26T13:09:02.1361563Z, CompileDate 2021-07-03T08:38:43.4120873Z, CreationDate 2020-02-26T07:16:44.3135253Z, DownloadWithoutReinit false, HandleErrorsWithinBlock false, InterfaceModifiedDate 2020-02-26T12:49:56.0619358Z, IsConsistent true, IsIECCheckEnabled false, IsKnowHowProtected false, ISMultiInstanceCapable true, IsRetainMemResEnabled false, IsWriteProtected false, LibraryConformanceStatus Warning: The object contains access to global data blocks. Warning: The block contains direct access to inputs, outputs, bit memories, indirect access to the registry or indirect access to external memory areas that are unknown at the time of compilation., MemoryReserve 100, ModifiedDate 2020-02-26T13:09:02.1361563Z, ParameterModified 2020-02-26T07:16:44.3135253Z, PLCSimAdvancedSupport true, SetENOAutomatically false, StructureModified 2020-02-26T12:49:56.0619358Z, UDAEnableTagReadback false
   VAR
      VlvLiq2 : "fbValve_Solenoid";
   END_VAR
BEGIN

REGION Network 1
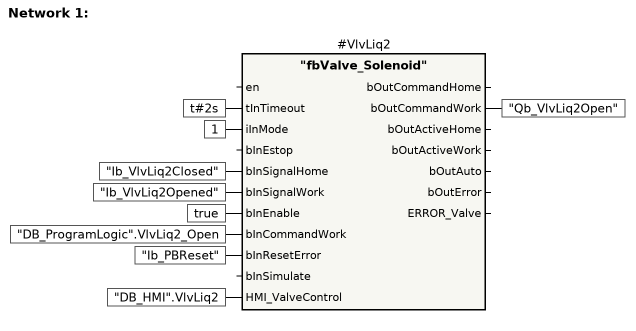
   #VlvLiq2(tInTimeout := t#2s,   // "fbValve_Solenoid"
            iInMode := 1,
            bInSignalHome := "Ib_VlvLiq2Closed",
            bInSignalWork := "Ib_VlvLiq2Opened",
            bInEnable := true,
            bInCommandWork := "DB_ProgramLogic".VlvLiq2_Open,
            bInResetError := "Ib_PBReset",
            HMI_ValveControl := "DB_HMI".VlvLiq2,
            bOutCommandWork => "Qb_VlvLiq2Open");
END_REGION
END_FUNCTION_BLOCK

FUNCTION_BLOCK "Program Logic"   // FB5, FBD
{ S7_Optimized_Access := 'TRUE' }
VERSION : 0.1
// stored: AutoNumber true, CodeModifiedDate 2020-02-26T12:59:57.0334412Z, CompileDate 2021-07-03T08:38:44.9588418Z, CreationDate 2020-02-26T07:17:15.9384502Z, DownloadWithoutReinit false, HandleErrorsWithinBlock false, InterfaceModifiedDate 2020-02-26T11:20:20.4837101Z, IsConsistent true, IsIECCheckEnabled false, IsKnowHowProtected false, ISMultiInstanceCapable true, IsRetainMemResEnabled false, IsWriteProtected false, LibraryConformanceStatus Warning: The object contains access to global data blocks. Warning: The block contains direct access to inputs, outputs, bit memories, indirect access to the registry or indirect access to external memory areas that are unknown at the time of compilation., MemoryReserve 100, ModifiedDate 2020-02-26T12:59:57.0334412Z, ParameterModified 2020-02-26T07:17:15.9384502Z, PLCSimAdvancedSupport true, SetENOAutomatically false, StructureModified 2020-02-26T11:20:20.4837101Z, UDAEnableTagReadback false
   VAR
      StepSeq : "fbStepSequencer";
      CurrentStep { S7_SetPoint := 'True'} : Int;
      NextStep : Int;
      StepDone : Bool;
   END_VAR
   VAR_TEMP   // added for the SCL form of the ladder/FBD networks
      _w1 : Bool;
   END_VAR
BEGIN

REGION Network 1: 0 -- Idle
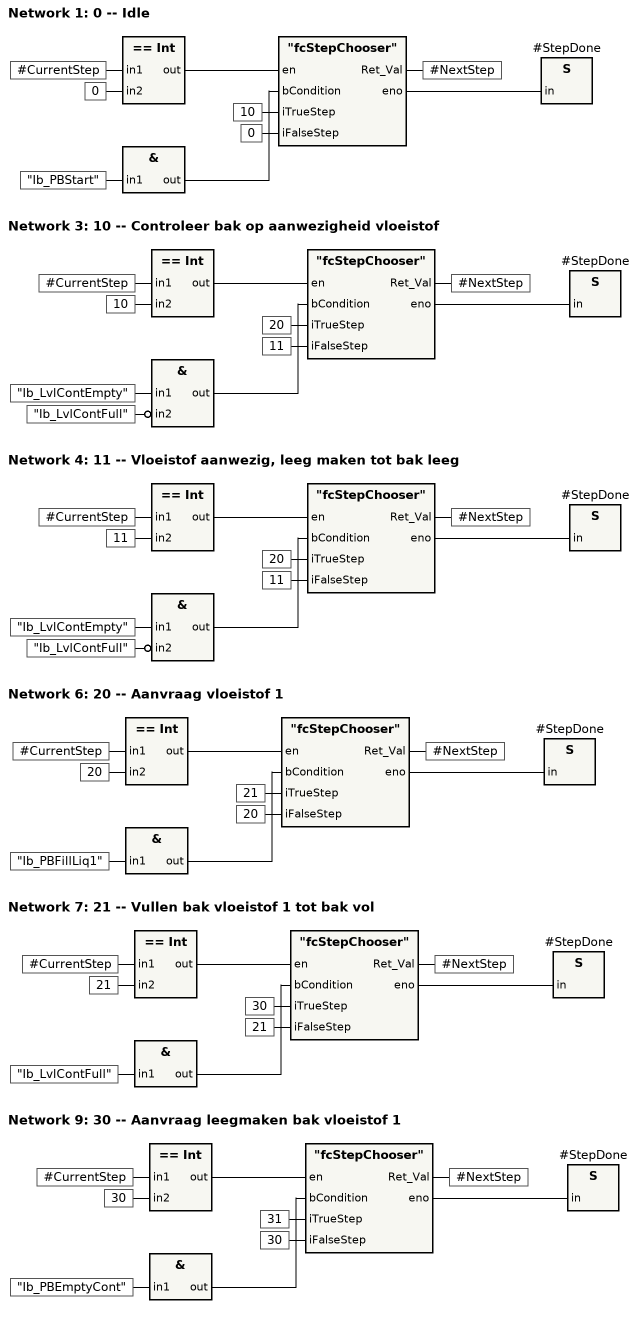
   #NextStep := "fcStepChooser"(EN := #CurrentStep = 0,
                           bCondition := "Ib_PBStart",
                           iTrueStep := 10,
                           iFalseStep := 0,
                           ENO => #_w1);
   IF #_w1 THEN #StepDone := TRUE; END_IF;
END_REGION

REGION Network 3: 10 -- Controleer bak op aanwezigheid vloeistof
   // vloeistof aanwezig 10->11
   // geen vloeistof aanwezig 10->20
   #NextStep := "fcStepChooser"(EN := #CurrentStep = 10,
                           bCondition := "Ib_LvlContEmpty" AND NOT "Ib_LvlContFull",
                           iTrueStep := 20,
                           iFalseStep := 11,
                           ENO => #_w1);
   IF #_w1 THEN #StepDone := TRUE; END_IF;
END_REGION

REGION Network 4: 11 -- Vloeistof aanwezig, leeg maken tot bak leeg
   #NextStep := "fcStepChooser"(EN := #CurrentStep = 11,
                           bCondition := "Ib_LvlContEmpty" AND NOT "Ib_LvlContFull",
                           iTrueStep := 20,
                           iFalseStep := 11,
                           ENO => #_w1);
   IF #_w1 THEN #StepDone := TRUE; END_IF;
END_REGION

REGION Network 6: 20 -- Aanvraag vloeistof 1
   #NextStep := "fcStepChooser"(EN := #CurrentStep = 20,
                           bCondition := "Ib_PBFillLiq1",
                           iTrueStep := 21,
                           iFalseStep := 20,
                           ENO => #_w1);
   IF #_w1 THEN #StepDone := TRUE; END_IF;
END_REGION

REGION Network 7: 21 -- Vullen bak vloeistof 1 tot bak vol
   #NextStep := "fcStepChooser"(EN := #CurrentStep = 21,
                           bCondition := "Ib_LvlContFull",
                           iTrueStep := 30,
                           iFalseStep := 21,
                           ENO => #_w1);
   IF #_w1 THEN #StepDone := TRUE; END_IF;
END_REGION

REGION Network 9: 30 -- Aanvraag leegmaken bak vloeistof 1
   #NextStep := "fcStepChooser"(EN := #CurrentStep = 30,
                           bCondition := "Ib_PBEmptyCont",
                           iTrueStep := 31,
                           iFalseStep := 30,
                           ENO => #_w1);
   IF #_w1 THEN #StepDone := TRUE; END_IF;
END_REGION

REGION Network 10: 31 -- Leeg maken bak vloeistof 1
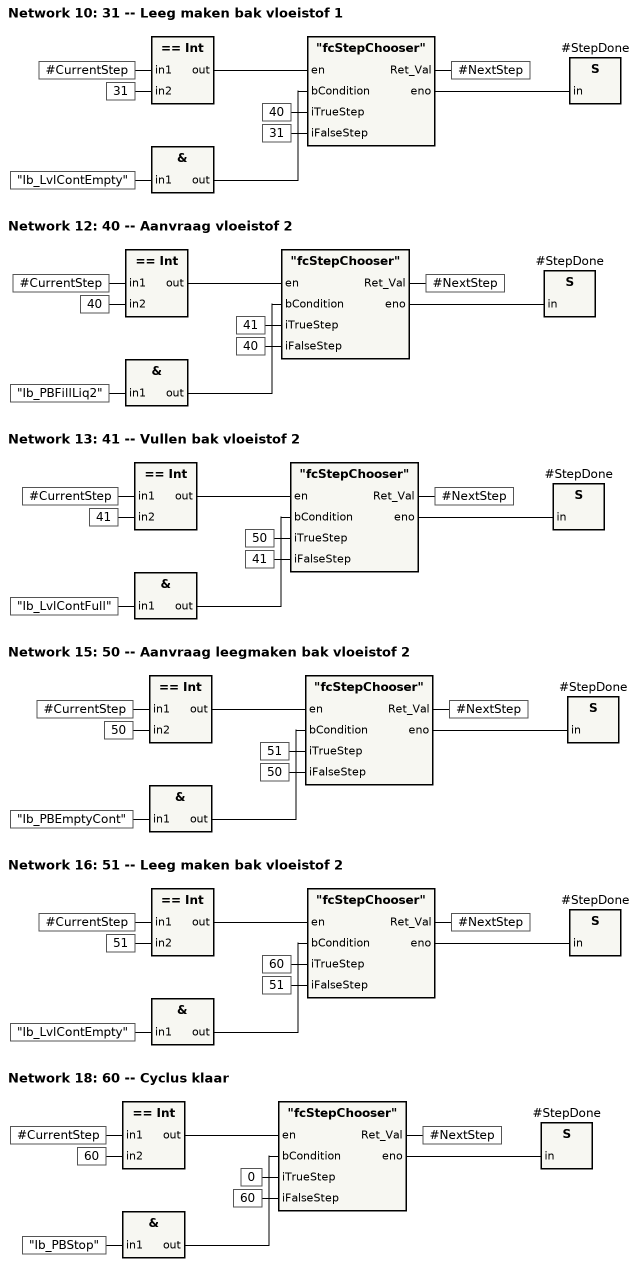
   #NextStep := "fcStepChooser"(EN := #CurrentStep = 31,
                           bCondition := "Ib_LvlContEmpty",
                           iTrueStep := 40,
                           iFalseStep := 31,
                           ENO => #_w1);
   IF #_w1 THEN #StepDone := TRUE; END_IF;
END_REGION

REGION Network 12: 40 -- Aanvraag vloeistof 2
   #NextStep := "fcStepChooser"(EN := #CurrentStep = 40,
                           bCondition := "Ib_PBFillLiq2",
                           iTrueStep := 41,
                           iFalseStep := 40,
                           ENO => #_w1);
   IF #_w1 THEN #StepDone := TRUE; END_IF;
END_REGION

REGION Network 13: 41 -- Vullen bak vloeistof 2
   #NextStep := "fcStepChooser"(EN := #CurrentStep = 41,
                           bCondition := "Ib_LvlContFull",
                           iTrueStep := 50,
                           iFalseStep := 41,
                           ENO => #_w1);
   IF #_w1 THEN #StepDone := TRUE; END_IF;
END_REGION

REGION Network 15: 50 -- Aanvraag leegmaken bak vloeistof 2
   #NextStep := "fcStepChooser"(EN := #CurrentStep = 50,
                           bCondition := "Ib_PBEmptyCont",
                           iTrueStep := 51,
                           iFalseStep := 50,
                           ENO => #_w1);
   IF #_w1 THEN #StepDone := TRUE; END_IF;
END_REGION

REGION Network 16: 51 -- Leeg maken bak vloeistof 2
   #NextStep := "fcStepChooser"(EN := #CurrentStep = 51,
                           bCondition := "Ib_LvlContEmpty",
                           iTrueStep := 60,
                           iFalseStep := 51,
                           ENO => #_w1);
   IF #_w1 THEN #StepDone := TRUE; END_IF;
END_REGION

REGION Network 18: 60 -- Cyclus klaar
   #NextStep := "fcStepChooser"(EN := #CurrentStep = 60,
                           bCondition := "Ib_PBStop",
                           iTrueStep := 0,
                           iFalseStep := 60,
                           ENO => #_w1);
   IF #_w1 THEN #StepDone := TRUE; END_IF;
END_REGION

REGION Network 20: Step Sequencer
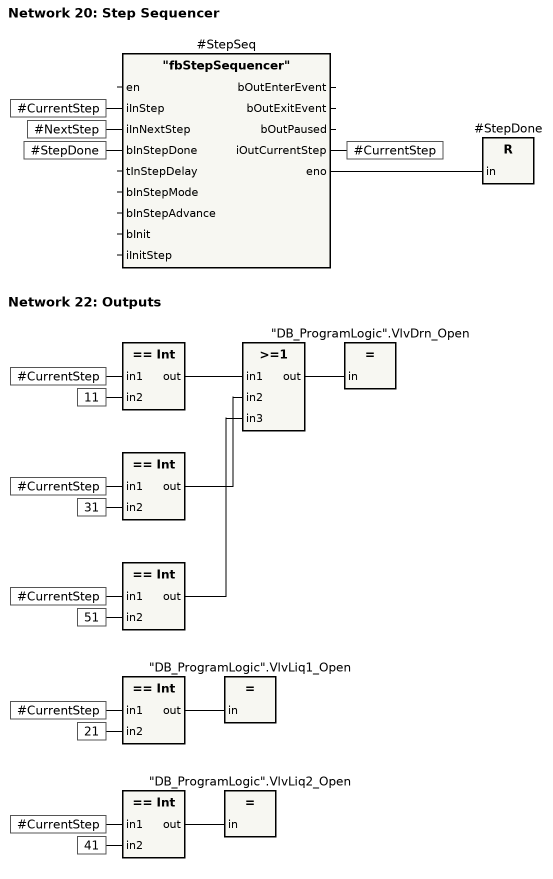
   #StepSeq(iInStep := #CurrentStep,   // "fbStepSequencer"
            iInNextStep := #NextStep,
            bInStepDone := #StepDone,
            iOutCurrentStep => #CurrentStep,
            ENO => #_w1);
   IF #_w1 THEN #StepDone := FALSE; END_IF;
END_REGION

REGION Network 22: Outputs
   "DB_ProgramLogic".VlvDrn_Open := (#CurrentStep = 11) OR (#CurrentStep = 31) OR (#CurrentStep = 51);
   "DB_ProgramLogic".VlvLiq1_Open := #CurrentStep = 21;
   "DB_ProgramLogic".VlvLiq2_Open := #CurrentStep = 41;
END_REGION
END_FUNCTION_BLOCK

FUNCTION "fcStepChooser" : Int   // FC185, SCL
{ S7_Optimized_Access := 'TRUE' }
VERSION : 0.0
// stored: AutoNumber false, CodeModifiedDate 2021-07-03T08:38:37.9433229Z, CompileDate 2021-07-03T08:38:37.9433229Z, CreationDate 2020-02-26T10:04:39.2339296Z, HandleErrorsWithinBlock false, InterfaceModifiedDate 2016-08-14T20:38:19.3457853Z, IsConsistent true, IsIECCheckEnabled false, IsKnowHowProtected false, IsWriteProtected false, LibraryConformanceStatus The object is library-conformant., LibraryType fcStepChooser V 3.0.1, LibraryTypeVersionGuid 8b64a3a6-6372-455a-bcc3-1a11207f1451, ModifiedDate 2021-07-03T08:38:37.9433229Z, ParameterModified 2016-08-14T20:38:19.3254825Z, PLCSimAdvancedSupport true, SetENOAutomatically true, StructureModified 2016-08-14T20:38:19.3457853Z, UDAEnableTagReadback false
   VAR_INPUT
      bCondition : Bool;
      iTrueStep : Int;
      iFalseStep : Int;
   END_VAR
   VAR_TEMP
      iResult : Int;
   END_VAR
BEGIN

       IF #bCondition THEN
           #iResult:=#iTrueStep;
       ELSE
           #iResult:=#iFalseStep;
       END_IF;
       ENO:=true;
       #fcStepChooser:=#iResult;
END_FUNCTION

FUNCTION_BLOCK "fbStepSequencer"   // FB185, SCL
TITLE = Step sequence controller
{ S7_Optimized_Access := 'TRUE' }
AUTHOR : Boris
VERSION : 4.0
// Modified by Ken Brey 2010-08-25 KLB.  Added Initialization inputs and logic.
// Modified by Ken Brey 2006-08-08 Removed initialization of inputs.  Initializing inputs doesn't do anything.  The input value if un-wired will be the last value
//                                   set for that input in a different call.  The initialized value in the declaration section does not set it back to default
//                                   if unwired.  Allways supply values for all inputs.
// Modified by Tim Jager 2005-12-13 no block Id in error message
// Modified by Boris: branched -> simplified version, no errors, no timeout; still have to use static memory for TON/CurStep (might be fixed later using in/out structure)
// Modified by Nick Shea:  2012-03-30 Re-instated step mode
// stored: AutoNumber false, CodeModifiedDate 2021-07-03T08:38:43.5995384Z, CompileDate 2021-07-03T08:38:43.5995384Z, CreationDate 2020-02-26T09:46:55.060709Z, DownloadWithoutReinit false, HandleErrorsWithinBlock false, InterfaceModifiedDate 2017-09-27T20:53:33.4400806Z, IsConsistent true, IsIECCheckEnabled false, IsKnowHowProtected false, ISMultiInstanceCapable true, IsRetainMemResEnabled false, IsWriteProtected false, LibraryConformanceStatus The object is library-conformant., LibraryType fbStepSequencer V 3.0.1, LibraryTypeVersionGuid beea64d7-3359-4773-b63d-f289c4512550, MemoryReserve 100, ModifiedDate 2021-07-03T08:38:43.5995384Z, ParameterModified 2016-08-14T20:38:38.9589289Z, PLCSimAdvancedSupport true, SetENOAutomatically true, StructureModified 2016-08-14T20:38:38.9704141Z, UDAEnableTagReadback false
   VAR_INPUT
      iInStep { ExternalAccessible := 'False'; ExternalVisible := 'False'; ExternalWritable := 'False'} : Int;   // Constant: current step required for the FB to run
      iInNextStep { ExternalAccessible := 'False'; ExternalVisible := 'False'; ExternalWritable := 'False'} : Int;   // Next step to go to if step is done
      bInStepDone { ExternalAccessible := 'False'; ExternalVisible := 'False'; ExternalWritable := 'False'} : Bool;   // if step done logic is true, then we move from IN_STEP to NEXT_STEP
      tInStepDelay { ExternalAccessible := 'False'; ExternalVisible := 'False'; ExternalWritable := 'False'} : Time;   // After the step done input is true, we wait for x seconds before moving to next
      bInStepMode { ExternalAccessible := 'False'; ExternalVisible := 'False'; ExternalWritable := 'False'} : Bool;   // Pause sequence at completion of current step
      bInStepAdvance { ExternalAccessible := 'False'; ExternalVisible := 'False'; ExternalWritable := 'False'} : Bool;   // If paused, trigger next step
      bInit { ExternalAccessible := 'False'; ExternalVisible := 'False'; ExternalWritable := 'False'} : Bool;
      iInitStep { ExternalAccessible := 'False'; ExternalVisible := 'False'; ExternalWritable := 'False'} : Int;
   END_VAR
   VAR_OUTPUT
      bOutEnterEvent { ExternalAccessible := 'False'; ExternalVisible := 'False'; ExternalWritable := 'False'} : Bool;
      bOutExitEvent { ExternalAccessible := 'False'; ExternalVisible := 'False'; ExternalWritable := 'False'} : Bool;
      bOutPaused { ExternalAccessible := 'False'; ExternalVisible := 'False'; ExternalWritable := 'False'} : Bool;   // Sequence is currently paused.
      iOutCurrentStep { ExternalAccessible := 'False'; ExternalVisible := 'False'; ExternalWritable := 'False'} : Int;   // output current step
   END_VAR
   VAR
      TON_StepDelay { ExternalAccessible := 'False'; ExternalVisible := 'False'; ExternalWritable := 'False'; S7_SetPoint := 'True'} : TON_TIME;   // used to delay moving to the next step.
      iCurrentStep { ExternalAccessible := 'False'; ExternalVisible := 'False'; ExternalWritable := 'False'} : Int;   // Current step of the sequencer
      bAlreadyInThisStep { ExternalAccessible := 'False'; ExternalVisible := 'False'; ExternalWritable := 'False'} : Bool;
   END_VAR
   VAR_TEMP
      bNoStepDelay : Bool;   // step delay disabled
   END_VAR
BEGIN


   //*****************************************************************************************
   // INSTRUCTION SECTION
   ENO:=false; //init variables
   #bOutExitEvent :=false;
   #bOutEnterEvent:=false;

   IF (#iInStep=#iCurrentStep) THEN
       IF NOT #bAlreadyInThisStep THEN
           #bOutEnterEvent:=true;
           #bAlreadyInThisStep:=true;
       END_IF;
       IF #bInStepDone THEN
           //Run Step done Timer
           #TON_StepDelay(IN:=(TRUE),PT:=#tInStepDelay);

           //check if we are using a step delay
           #bNoStepDelay:= (#tInStepDelay<=T#0MS);

           //We can move to the next step if (STEP_DONE and StepDelay timer complete) 
           //  AND
           //(we are in step mode and the step advance is true, or if we are not in step mode 
           //  AND
           //It is not the first scan of this step
           IF ((#TON_StepDelay.Q OR #bNoStepDelay) AND (NOT #bInStepMode OR (#bInStepMode AND #bInStepAdvance)) AND NOT #bOutEnterEvent) THEN 
               #iCurrentStep   := #iInNextStep;   //move to next step
               //Reset Step done Timer
               #TON_StepDelay(IN:=(false),PT:=#tInStepDelay); 
               #bOutExitEvent:=true;
               #bAlreadyInThisStep:=false;
           END_IF;
       END_IF;
       #bOutPaused := #bInStepDone AND (#TON_StepDelay.Q OR #bNoStepDelay) AND (#bInStepMode AND NOT #bInStepAdvance);
       //Only set this if we are ok and in the right step
       ENO:= true;
   END_IF;
   IF (#bInit) THEN
       #iCurrentStep := #iInitStep;
       #bInit:=false;  //Clear so that if it is unwired on the next call, it is not run.
       #bAlreadyInThisStep:=false;
   END_IF;

   //Set output variables
   #iOutCurrentStep := #iCurrentStep;
   #tInStepDelay := T#0MS;
END_FUNCTION_BLOCK

DATA_BLOCK "Program Logic_DB"   // DB2
{ S7_Optimized_Access := 'TRUE' }
VERSION : 0.1
// stored: AutoNumber true, CodeModifiedDate 2020-02-26T12:50:20.2800962Z, CompileDate 2021-07-03T08:38:45.0845051Z, CreationDate 2020-02-26T12:50:20.1014064Z, DBAccessibleFromOPCUA true, DownloadWithoutReinit false, InstanceOfName Program Logic, InstanceOfNumber 5, InstanceOfType FB, InterfaceModifiedDate 2020-02-26T11:20:20.4837101Z, IsConsistent true, IsKnowHowProtected false, IsRetainMemResEnabled false, MemoryReserve 100, ModifiedDate 2020-02-26T12:50:20.2800962Z, ParameterModified 2020-02-26T07:17:15.9384502Z, StructureModified 2020-02-26T11:20:20.4837101Z, UDAEnableTagReadback false
"Program Logic"
BEGIN
END_DATA_BLOCK

DATA_BLOCK "Valve Drain_DB"   // DB7
{ S7_Optimized_Access := 'TRUE' }
VERSION : 0.1
// stored: AutoNumber true, CodeModifiedDate 2020-02-26T12:49:16.2970167Z, CompileDate 2021-07-03T08:38:43.5846302Z, CreationDate 2020-02-26T12:48:12.3344036Z, DBAccessibleFromOPCUA true, DownloadWithoutReinit false, InstanceOfName Valve Drain, InstanceOfNumber 4, InstanceOfType FB, InterfaceModifiedDate 2020-02-26T12:48:59.514304Z, IsConsistent true, IsKnowHowProtected false, IsRetainMemResEnabled false, MemoryReserve 100, ModifiedDate 2020-02-26T12:49:16.2970167Z, ParameterModified 2020-02-26T07:16:51.9541274Z, StructureModified 2020-02-26T12:48:59.514304Z, UDAEnableTagReadback false
"Valve Drain"
BEGIN
END_DATA_BLOCK

DATA_BLOCK "Valve Liquid 1_DB"   // DB8
{ S7_Optimized_Access := 'TRUE' }
VERSION : 0.1
// stored: AutoNumber true, CodeModifiedDate 2020-02-26T12:49:41.2445202Z, CompileDate 2021-07-03T08:38:43.2873738Z, CreationDate 2020-02-26T12:48:17.7591506Z, DBAccessibleFromOPCUA true, DownloadWithoutReinit false, InstanceOfName Valve Liquid 1, InstanceOfNumber 2, InstanceOfType FB, InterfaceModifiedDate 2020-02-26T12:49:32.479094Z, IsConsistent true, IsKnowHowProtected false, IsRetainMemResEnabled false, MemoryReserve 100, ModifiedDate 2020-02-26T12:49:41.2445202Z, ParameterModified 2020-02-26T07:16:31.1886327Z, StructureModified 2020-02-26T12:49:32.479094Z, UDAEnableTagReadback false
"Valve Liquid 1"
BEGIN
END_DATA_BLOCK

DATA_BLOCK "Valve Liquid 2_DB"   // DB9
{ S7_Optimized_Access := 'TRUE' }
VERSION : 0.1
// stored: AutoNumber true, CodeModifiedDate 2020-02-26T12:50:04.6689241Z, CompileDate 2021-07-03T08:38:43.4588479Z, CreationDate 2020-02-26T12:48:33.7755421Z, DBAccessibleFromOPCUA true, DownloadWithoutReinit false, InstanceOfName Valve Liquid 2, InstanceOfNumber 3, InstanceOfType FB, InterfaceModifiedDate 2020-02-26T12:49:56.0619358Z, IsConsistent true, IsKnowHowProtected false, IsRetainMemResEnabled false, MemoryReserve 100, ModifiedDate 2020-02-26T12:50:04.6689241Z, ParameterModified 2020-02-26T07:16:44.3135253Z, StructureModified 2020-02-26T12:49:56.0619358Z, UDAEnableTagReadback false
"Valve Liquid 2"
BEGIN
END_DATA_BLOCK
